	REGION J1.11.1
	    //J1.11.1
	    #"J1.11.1"(ConveyorID := _."J1.11.1",
	               ConveyorSensor:=_."ASiGW-MCC001-bw143-C1: Input"."Sensor J1.11.7",
	               Fault := DB_UDI.EmptyLine.Fault.Stop.Conveyor[_."J1.11.1"],
	               Upstream := DB_UDI.EmptyLine.Upstream.Conveyor[_."J1.11.1"],
	               Downstream := DB_UDI.EmptyLine.DownstreamAcu.Stop.Conveyor[_."J1.11.1"],
	               Interlock := DB_UDI.EmptyLine.Interlock.Stop.Conveyor[_."J1.11.1"],
	               RunForward => _."ASiGW-MCC001-bw143-C1: Output"."Motor J1.11.1",
	               WriteAsiDir => _."ASiGW-MCC001-bw143-C1: Output"."Dir J1.11.1");
	    
	END_REGION
	
	REGION J1.11.2
	    //J1.11.2
	    #"J1.11.2"(ConveyorID:=_."J1.11.2",
	               ConveyorSensor:=_."ASiGW-MCC001-bw143-C1: Input"."Sensor J1.11.7",
	                   Fault:= DB_UDI.EmptyLine.Fault.Stop.Conveyor[_."J1.11.2"],
	                   Upstream:= DB_UDI.EmptyLine.Upstream.Conveyor[_."J1.11.2"],
	                   Downstream:= DB_UDI.EmptyLine.DownstreamAcu.Stop.Conveyor[_."J1.11.2"],
	                   Interlock:= DB_UDI.EmptyLine.Interlock.Stop.Conveyor[_."J1.11.2"],
	                   RunForward => _."ASiGW-MCC001-bw143-C1: Output"."Motor J1.11.2",
	                   WriteAsiDir => _."ASiGW-MCC001-bw143-C1: Output"."Dir J1.11.2");
	
	END_REGION
	
	REGION J1.11.3
	    //J1.11.3
	    #"J1.11.3"(ConveyorID:=_."J1.11.3",
	               ConveyorSensor:=_."ASiGW-MCC001-bw143-C1: Input"."Sensor J1.11.7",
	                   Fault:= DB_UDI.EmptyLine.Fault.Stop.Conveyor[_."J1.11.3"],
	                   Upstream:= DB_UDI.EmptyLine.Upstream.Conveyor[_."J1.11.3"],
	                   Downstream:= DB_UDI.EmptyLine.DownstreamAcu.Stop.Conveyor[_."J1.11.3"],
	                   Interlock:= DB_UDI.EmptyLine.Interlock.Stop.Conveyor[_."J1.11.3"],
	                   RunForward => _."ASiGW-MCC001-bw143-C1: Output"."Motor J1.11.3",
	                   WriteAsiDir => _."ASiGW-MCC001-bw143-C1: Output"."Dir J1.11.3");
	
	END_REGION
	
	REGION J1.11.4
	    //J1.11.4
	    #"J1.11.4"(ConveyorID := _."J1.11.4",
	               ConveyorSensor:=_."ASiGW-MCC001-bw143-C1: Input"."Sensor J1.11.7",
	               Fault := DB_UDI.EmptyLine.Fault.Stop.Conveyor[_."J1.11.4"],
	               Upstream := DB_UDI.EmptyLine.Upstream.Conveyor[_."J1.11.4"],
	               Downstream := DB_UDI.EmptyLine.DownstreamAcu.Stop.Conveyor[_."J1.11.4"],
	               Interlock := DB_UDI.EmptyLine.Interlock.Stop.Conveyor[_."J1.11.4"],
	               RunForward => _."ASiGW-MCC001-bw143-C1: Output"."Motor J1.11.4",
	               WriteAsiDir => _."ASiGW-MCC001-bw143-C1: Output"."Dir J1.11.4");
	    
	END_REGION
	
	REGION J1.11.5
	    //J1.11.5
	    #"J1.11.5"(ConveyorID:=_."J1.11.5",
	               ConveyorSensor:=_."ASiGW-MCC001-bw143-C1: Input"."Sensor J1.11.7",
	                   Fault:= DB_UDI.EmptyLine.Fault.Stop.Conveyor[_."J1.11.5"],
	                   Upstream:= DB_UDI.EmptyLine.Upstream.Conveyor[_."J1.11.5"],
	                   Downstream:= DB_UDI.EmptyLine.DownstreamAcu.Stop.Conveyor[_."J1.11.5"],
	                   Interlock:= DB_UDI.EmptyLine.Interlock.Stop.Conveyor[_."J1.11.5"],
	                   RunForward => _."ASiGW-MCC001-bw143-C1: Output"."Motor J1.11.5",
	                   WriteAsiDir => _."ASiGW-MCC001-bw143-C1: Output"."Dir J1.11.5");
	
	END_REGION
	
	REGION J1.11.6
	    //J1.11.6
	    #"J1.11.6"(ConveyorID := _."J1.11.6",
	               ConveyorSensor:=_."ASiGW-MCC001-bw143-C1: Input"."Sensor J1.11.7",
	               Fault := DB_UDI.EmptyLine.Fault.Stop.Conveyor[_."J1.11.6"],
	               Upstream := DB_UDI.EmptyLine.Upstream.Conveyor[_."J1.11.6"],
	               Downstream := DB_UDI.EmptyLine.DownstreamAcu.Stop.Conveyor[_."J1.11.6"],
	               Interlock := DB_UDI.EmptyLine.Interlock.Stop.Conveyor[_."J1.11.6"],
	               RunForward => _."ASiGW-MCC001-bw143-C1: Output"."Motor J1.11.6",
	               WriteAsiDir => _."ASiGW-MCC001-bw143-C1: Output"."Dir J1.11.6");
	    
	END_REGION
	
	REGION J1.11.7
	    //J1.11.7
	    #"J1.11.7"(ConveyorID := _."J1.11.7",
	               ConveyorSensor:=_."ASiGW-MCC001-bw143-C1: Input"."Sensor J1.11.7",
	               Fault := DB_UDI.EmptyLine.Fault.Stop.Conveyor[_."J1.11.7"],
	               Upstream := DB_UDI.EmptyLine.Upstream.Conveyor[_."J1.11.7"],
	               Downstream := DB_UDI.EmptyLine.DownstreamAcu.Stop.Conveyor[_."J1.11.7"],
	               Interlock := DB_UDI.EmptyLine.Interlock.Stop.Conveyor[_."J1.11.7"],
	               RunForward => _."ASiGW-MCC001-bw143-C1: Output"."Motor J1.11.9",
	               WriteAsiDir => _."ASiGW-MCC001-bw143-C1: Output"."Dir J1.11.9");
	    
	END_REGION
	
	REGION J1.11.8
	    //J1.11.8
	    #"J1.11.8"(ConveyorID := _."J1.11.8",
	               ConveyorSensor:=_."ASiGW-MCC001-bw143-C1: Input"."Sensor J1.11.13",
	               Fault := DB_UDI.EmptyLine.Fault.Stop.Conveyor[_."J1.11.8"],
	               Upstream := DB_UDI.EmptyLine.Upstream.Conveyor[_."J1.11.8"],
	               Downstream := DB_UDI.EmptyLine.DownstreamAcu.Stop.Conveyor[_."J1.11.8"],
	               Interlock := DB_UDI.EmptyLine.Interlock.Stop.Conveyor[_."J1.11.8"],
	               RunForward => _."ASiGW-MCC001-bw143-C1: Output"."Motor J1.11.10",
	               WriteAsiDir => _."ASiGW-MCC001-bw143-C1: Output"."Dir J1.11.10");
	    
	END_REGION
	
	REGION J1.11.9
	    //J1.11.9
	    #"J1.11.9"(ConveyorID:=_."J1.11.9",
	               ConveyorSensor:=_."ASiGW-MCC001-bw143-C1: Input"."Sensor J1.11.13",
	                   Fault:= DB_UDI.EmptyLine.Fault.Stop.Conveyor[_."J1.11.9"],
	                   Upstream:= DB_UDI.EmptyLine.Upstream.Conveyor[_."J1.11.9"],
	                   Downstream:= DB_UDI.EmptyLine.DownstreamAcu.Stop.Conveyor[_."J1.11.9"],
	                   Interlock:= DB_UDI.EmptyLine.Interlock.Stop.Conveyor[_."J1.11.9"],
	                   RunForward => _."ASiGW-MCC001-bw143-C1: Output"."Motor J1.11.11",
	                   WriteAsiDir => _."ASiGW-MCC001-bw143-C1: Output"."Dir J1.11.11");
	        
	END_REGION
	
	REGION J1.11.10
	    //J1.11.10
	    #"J1.11.10"(ConveyorID:=_."J1.11.10",
	                ConveyorSensor:=_."ASiGW-MCC001-bw143-C1: Input"."Sensor J1.11.13",
	                   Fault:= DB_UDI.EmptyLine.Fault.Stop.Conveyor[_."J1.11.10"],
	                   Upstream:= DB_UDI.EmptyLine.Upstream.Conveyor[_."J1.11.10"],
	                   Downstream:= DB_UDI.EmptyLine.DownstreamAcu.Stop.Conveyor[_."J1.11.10"],
	                   Interlock:= DB_UDI.EmptyLine.Interlock.Stop.Conveyor[_."J1.11.10"],
	                   RunForward => _."ASiGW-MCC001-bw143-C1: Output"."Motor J1.11.12",
	                   WriteAsiDir => _."ASiGW-MCC001-bw143-C1: Output"."Dir J1.11.12");
	
	END_REGION
	
	REGION J1.11.11
	    //J1.11.11
	    #"J1.11.11"(ConveyorID:=_."J1.11.11",
	                ConveyorSensor:=_."ASiGW-MCC001-bw143-C1: Input"."Sensor J1.11.13",
	                   Fault:= DB_UDI.EmptyLine.Fault.Stop.Conveyor[_."J1.11.11"],
	                   Upstream:= DB_UDI.EmptyLine.Upstream.Conveyor[_."J1.11.11"],
	                   Downstream:= DB_UDI.EmptyLine.DownstreamAcu.Stop.Conveyor[_."J1.11.11"],
	                   Interlock:= DB_UDI.EmptyLine.Interlock.Stop.Conveyor[_."J1.11.11"],
	                   RunForward => _."ASiGW-MCC001-bw143-C1: Output"."Motor J1.11.13",
	                   WriteAsiDir => _."ASiGW-MCC001-bw143-C1: Output"."Dir J1.11.13");
	
	END_REGION
	
	REGION J1.11.12
	    //J1.11.12
	    #"J1.11.12"(ConveyorID := _."J1.11.12",
	                ConveyorSensor:=_."ASiGW-MCC001-bw143-C1: Input"."Sensor J1.11.13",
	                Fault := DB_UDI.EmptyLine.Fault.Stop.Conveyor[_."J1.11.12"],
	                Upstream := DB_UDI.EmptyLine.Upstream.Conveyor[_."J1.11.12"],
	                Downstream := DB_UDI.EmptyLine.DownstreamAcu.Stop.Conveyor[_."J1.11.12"],
	                Interlock := DB_UDI.EmptyLine.Interlock.Stop.Conveyor[_."J1.11.12"],
	                RunForward => _."ASiGW-MCC001-bw143-C1: Output"."Motor J1.11.12",
	                WriteAsiDir => _."ASiGW-MCC001-bw143-C1: Output"."Dir J1.11.12");
	    
	END_REGION
	
	REGION J1.11.13
	    //J1.11.13
	    #"J1.11.13"(ConveyorID:=_."J1.11.13",
	                ConveyorSensor:=_."ASiGW-MCC001-bw143-C1: Input"."Sensor J1.11.13",
	                   Fault:= DB_UDI.EmptyLine.Fault.Stop.Conveyor[_."J1.11.13"],
	                   Upstream:= DB_UDI.EmptyLine.Upstream.Conveyor[_."J1.11.13"],
	                   Downstream:= DB_UDI.EmptyLine.DownstreamAcu.Stop.Conveyor[_."J1.11.13"],
	                   Interlock:= DB_UDI.EmptyLine.Interlock.Stop.Conveyor[_."J1.11.13"],
	                   RunForward => _."ASiGW-MCC001-bw143-C1: Output"."Motor J1.11.13",
	                   WriteAsiDir => _."ASiGW-MCC001-bw143-C1: Output"."Dir J1.11.13");
	
	END_REGION
	
	REGION K1.1.1
	    //K1.1.1  (Go Left)
	    #"K1.1.1"(ConveyorID:=_."K1.1.1",
	              ConveyorSensor:=_."ASiGW-MCC001-bw143-C2: Input"."Sensor K1.2.1",
	                   Fault:= DB_UDI.EmptyLine.Fault.Stop.Conveyor[_."K1.1.1"],
	                   Upstream:= DB_UDI.EmptyLine.Upstream.Conveyor[_."K1.1.1"],
	                   Downstream:= DB_UDI.EmptyLine.DownstreamAcu.Stop.Conveyor[_."K1.1.1"],
	                   Interlock:= DB_UDI.EmptyLine.Interlock.Stop.Conveyor[_."K1.1.1"],
	                   RunForward => _."ASiGW-MCC001-bw143-C2: Output"."Motor K1.1.1",
	                   WriteAsiDir => _."ASiGW-MCC001-bw143-C2: Output"."Dir K1.1.1");
	         
	END_REGION
	
	REGION K1.2.1
	    //K1.2.1
	    #"K1.2.1"(ConveyorID:=_."K1.2.1",
	              ConveyorSensor:=_."ASiGW-MCC001-bw143-C2: Input"."Sensor K1.2.1",
	                   Fault:= DB_UDI.EmptyLine.Fault.Stop.Conveyor[_."K1.2.1"],
	                   Upstream:= DB_UDI.EmptyLine.Upstream.Conveyor[_."K1.2.1"],
	                   Downstream:= DB_UDI.EmptyLine.DownstreamAcu.Stop.Conveyor[_."K1.2.1"],
	                   Interlock:= DB_UDI.EmptyLine.Interlock.Stop.Conveyor[_."K1.2.1"],
	                   RunForward => _."ASiGW-MCC001-bw143-C2: Output"."Motor - K1.2.1",
	                   WriteAsiDir => _."ASiGW-MCC001-bw143-C2: Output"."2-31A Dir",
	                   WriteAsiSpeed=>_."ASiGW-MCC001-bw143-C2: Output"."2-31A Speed");
	         
	END_REGION
	
	REGION K1.3.1
	    //K1.3.1
	    #"K1.3.1"(ConveyorID := _."K1.3.1",
	              ConveyorSensor:=_."ASiGW-MCC001-bw143-C2: Input"."Sensor K1.3.1",
	              Fault := DB_UDI.EmptyLine.Fault.Stop.Conveyor[_."K1.3.1"],
	              Upstream := DB_UDI.EmptyLine.Upstream.Conveyor[_."K1.3.1"],
	              Downstream := DB_UDI.EmptyLine.DownstreamAcu.Stop.Conveyor[_."K1.3.1"],
	              Interlock := DB_UDI.EmptyLine.Interlock.Stop.Conveyor[_."K1.3.1"],
	              RunForward => _."ASiGW-MCC001-bw143-C2: Output"."Motor K1.3.1",
	              WriteAsiDir => _."ASiGW-MCC001-bw143-C2: Output"."Dir K1.3.1");
	    
	END_REGION
	
	REGION K1.4.1
	    //K1.4.1
	    #"K1.4.1"(ConveyorID:=_."K1.4.1",
	              ConveyorSensor:=_."ASiGW-MCC001-bw143-C2: Input"."Sensor K1.4.1",
	                   Fault:= DB_UDI.EmptyLine.Fault.Stop.Conveyor[_."K1.4.1"],
	                   Upstream:= DB_UDI.EmptyLine.Upstream.Conveyor[_."K1.4.1"],
	                   Downstream:= DB_UDI.EmptyLine.DownstreamAcu.Stop.Conveyor[_."K1.4.1"],
	                   Interlock:= DB_UDI.EmptyLine.Interlock.Stop.Conveyor[_."K1.4.1"],
	                   RunForward => _."ASiGW-MCC001-bw143-C2: Output"."Motor K1.4.1",
	                   WriteAsiDir => _."ASiGW-MCC001-bw143-C2: Output"."Dir K1.4.1");
	         
	END_REGION
	
	REGION K1.4.2
	    //K1.4.2
	    #"K1.4.2"(ConveyorID := _."K1.4.2",
	              ConveyorSensor:=_."ASiGW-MCC001-bw143-C2: Input"."Sensor K1.4.10",
	              Fault := DB_UDI.EmptyLine.Fault.Stop.Conveyor[_."K1.4.2"],
	              Upstream := DB_UDI.EmptyLine.Upstream.Conveyor[_."K1.4.2"],
	              Downstream := DB_UDI.EmptyLine.DownstreamAcu.Stop.Conveyor[_."K1.4.2"],
	              Interlock := DB_UDI.EmptyLine.Interlock.Stop.Conveyor[_."K1.4.2"],
	              RunForward => _."ASiGW-MCC001-bw143-C2: Output"."Motor K1.4.2",
	              WriteAsiDir => _."ASiGW-MCC001-bw143-C2: Output"."Dir K1.4.2");
	    
	END_REGION
	
	REGION K1.4.3
	    //K1.4.3
	    #"K1.4.3"(ConveyorID := _."K1.4.3",
	              ConveyorSensor:=_."ASiGW-MCC001-bw143-C2: Input"."Sensor K1.4.10",
	              Fault := DB_UDI.EmptyLine.Fault.Stop.Conveyor[_."K1.4.3"],
	              Upstream := DB_UDI.EmptyLine.Upstream.Conveyor[_."K1.4.3"],
	              Downstream := DB_UDI.EmptyLine.DownstreamAcu.Stop.Conveyor[_."K1.4.3"],
	              Interlock := DB_UDI.EmptyLine.Interlock.Stop.Conveyor[_."K1.4.3"],
	              RunForward => _."ASiGW-MCC001-bw143-C2: Output"."Motor K1.4.3",
	              WriteAsiDir => _."ASiGW-MCC001-bw143-C2: Output"."Dir K1.4.3");
	    
	END_REGION
	
	REGION K1.4.4
	    //K1.4.4
	    #"K1.4.4"(ConveyorID := _."K1.4.4",
	              ConveyorSensor:=_."ASiGW-MCC001-bw143-C2: Input"."Sensor K1.4.10",
	              Fault := DB_UDI.EmptyLine.Fault.Stop.Conveyor[_."K1.4.4"],
	              Upstream := DB_UDI.EmptyLine.Upstream.Conveyor[_."K1.4.4"],
	              Downstream := DB_UDI.EmptyLine.DownstreamAcu.Stop.Conveyor[_."K1.4.4"],
	              Interlock := DB_UDI.EmptyLine.Interlock.Stop.Conveyor[_."K1.4.4"],
	              RunForward => _."ASiGW-MCC001-bw143-C2: Output"."Motor K1.4.4",
	              WriteAsiDir => _."ASiGW-MCC001-bw143-C2: Output"."Dir K1.4.4");
	    
	END_REGION
	
	REGION K1.4.5
	    //K1.4.5
	    #"K1.4.5"(ConveyorID := _."K1.4.5",
	              ConveyorSensor:=_."ASiGW-MCC001-bw143-C2: Input"."Sensor K1.4.10",
	              Fault := DB_UDI.EmptyLine.Fault.Stop.Conveyor[_."K1.4.5"],
	              Upstream := DB_UDI.EmptyLine.Upstream.Conveyor[_."K1.4.5"],
	              Downstream := DB_UDI.EmptyLine.DownstreamAcu.Stop.Conveyor[_."K1.4.5"],
	              Interlock := DB_UDI.EmptyLine.Interlock.Stop.Conveyor[_."K1.4.5"],
	              RunForward => _."ASiGW-MCC001-bw143-C2: Output"."Motor K1.4.5",
	              WriteAsiDir => _."ASiGW-MCC001-bw143-C2: Output"."Dir K1.4.5");
	    
	END_REGION
	
	REGION K1.4.6
	    //K1.4.6
	    #"K1.4.6"(ConveyorID:=_."K1.4.6",
	              ConveyorSensor:=_."ASiGW-MCC001-bw143-C2: Input"."Sensor K1.4.10",
	                   Fault:= DB_UDI.EmptyLine.Fault.Stop.Conveyor[_."K1.4.6"],
	                   Upstream:= DB_UDI.EmptyLine.Upstream.Conveyor[_."K1.4.6"],
	                   Downstream:= DB_UDI.EmptyLine.DownstreamAcu.Stop.Conveyor[_."K1.4.6"],
	                   Interlock:= DB_UDI.EmptyLine.Interlock.Stop.Conveyor[_."K1.4.6"],
	                   RunForward => _."ASiGW-MCC001-bw143-C2: Output"."Motor K1.4.6",
	                   WriteAsiDir => _."ASiGW-MCC001-bw143-C2: Output"."Dir K1.4.6");
	         
	END_REGION
	
	REGION K1.4.7
	    //K1.4.7
	    #"K1.4.7"(ConveyorID := _."K1.4.7",
	              ConveyorSensor:=_."ASiGW-MCC001-bw143-C2: Input"."Sensor K1.4.10",
	              Fault := DB_UDI.EmptyLine.Fault.Stop.Conveyor[_."K1.4.7"],
	              Upstream := DB_UDI.EmptyLine.Upstream.Conveyor[_."K1.4.7"],
	              Downstream := DB_UDI.EmptyLine.DownstreamAcu.Stop.Conveyor[_."K1.4.7"],
	              Interlock := DB_UDI.EmptyLine.Interlock.Stop.Conveyor[_."K1.4.7"],
	              RunForward => _."ASiGW-MCC001-bw143-C2: Output"."Motor K1.4.7",
	              WriteAsiDir => _."ASiGW-MCC001-bw143-C2: Output"."Dir K1.4.7");
	    
	END_REGION
	
	REGION K1.4.8
	    //K1.4.8
	    #"K1.4.8"(ConveyorID := _."K1.4.8",
	              ConveyorSensor:=_."ASiGW-MCC001-bw143-C2: Input"."Sensor K1.4.10",
	              Fault := DB_UDI.EmptyLine.Fault.Stop.Conveyor[_."K1.4.8"],
	              Upstream := DB_UDI.EmptyLine.Upstream.Conveyor[_."K1.4.8"],
	              Downstream := DB_UDI.EmptyLine.DownstreamAcu.Stop.Conveyor[_."K1.4.8"],
	              Interlock := DB_UDI.EmptyLine.Interlock.Stop.Conveyor[_."K1.4.8"],
	              RunForward => _."ASiGW-MCC001-bw143-C2: Output"."Motor K1.4.8",
	              WriteAsiDir => _."ASiGW-MCC001-bw143-C2: Output"."Dir K1.4.8");
	    
	END_REGION
	
	REGION K1.4.9
	    //K1.4.9
	    #"K1.4.9"(ConveyorID:=_."K1.4.9",
	              ConveyorSensor:=_."ASiGW-MCC001-bw143-C2: Input"."Sensor K1.4.10",
	                   Fault:= DB_UDI.EmptyLine.Fault.Stop.Conveyor[_."K1.4.9"],
	                   Upstream:= DB_UDI.EmptyLine.Upstream.Conveyor[_."K1.4.9"],
	                   Downstream:= DB_UDI.EmptyLine.DownstreamAcu.Stop.Conveyor[_."K1.4.9"],
	                   Interlock:= DB_UDI.EmptyLine.Interlock.Stop.Conveyor[_."K1.4.9"],
	                   RunForward => _."ASiGW-MCC001-bw143-C2: Output"."Motor K1.4.9",
	                   WriteAsiDir => _."ASiGW-MCC001-bw143-C2: Output"."Dir K1.4.9");
	         
	END_REGION
	
	REGION K1.4.10
	    //K1.4.10
	    #"K1.4.10"(ConveyorID:=_."K1.4.10",
	               ConveyorSensor:=_."ASiGW-MCC001-bw143-C2: Input"."Sensor K1.4.10",
	                   Fault:= DB_UDI.EmptyLine.Fault.Stop.Conveyor[_."K1.4.10"],
	                   Upstream:= DB_UDI.EmptyLine.Upstream.Conveyor[_."K1.4.10"],
	                   Downstream:= DB_UDI.EmptyLine.DownstreamAcu.Stop.Conveyor[_."K1.4.10"],
	                   Interlock:= DB_UDI.EmptyLine.Interlock.Stop.Conveyor[_."K1.4.10"],
	                   RunForward => _."ASiGW-MCC001-bw143-C2: Output"."Motor K1.4.10",
	                   WriteAsiDir => _."ASiGW-MCC001-bw143-C2: Output"."Dir K1.4.10");
	        
	END_REGION
	
	REGION K1.5.1
	    //K1.5.1
	    #"K1.5.1"(ConveyorID:=_."K1.5.1",
	              ConveyorSensor:=_."ASiGW-MCC001-bw143-C2: Input"."Sensor K1.5.8",
	                   Fault:= DB_UDI.EmptyLine.Fault.Stop.Conveyor[_."K1.5.1"],
	                   Upstream:= DB_UDI.EmptyLine.Upstream.Conveyor[_."K1.5.1"],
	                   Downstream:= DB_UDI.EmptyLine.DownstreamAcu.Stop.Conveyor[_."K1.5.1"],
	                   Interlock:= DB_UDI.EmptyLine.Interlock.Stop.Conveyor[_."K1.5.1"],
	                   RunForward => _."ASiGW-MCC001-bw143-C2: Output"."Motor K1.5.1",
	                   WriteAsiDir => _."ASiGW-MCC001-bw143-C2: Output"."Dir K1.5.1");
	
	END_REGION
	
	REGION K1.5.2
	    //K1.5.2
	    #"K1.5.2"(ConveyorID:=_."K1.5.2",
	              ConveyorSensor:=_."ASiGW-MCC001-bw143-C2: Input"."Sensor K1.5.8",
	                   Fault:= DB_UDI.EmptyLine.Fault.Stop.Conveyor[_."K1.5.2"],
	                   Upstream:= DB_UDI.EmptyLine.Upstream.Conveyor[_."K1.5.2"],
	                   Downstream:= DB_UDI.EmptyLine.DownstreamAcu.Stop.Conveyor[_."K1.5.2"],
	                   Interlock:= DB_UDI.EmptyLine.Interlock.Stop.Conveyor[_."K1.5.2"],
	                   RunForward => _."ASiGW-MCC001-bw143-C2: Output"."Motor K1.5.2",
	                   WriteAsiDir => _."ASiGW-MCC001-bw143-C2: Output"."Dir K1.5.2");
	         
	
	END_REGION
	
	REGION K1.5.3
	    //K1.5.3
	    #"K1.5.3"(ConveyorID:=_."K1.5.3",
	              ConveyorSensor:=_."ASiGW-MCC001-bw143-C2: Input"."Sensor K1.5.8",
	                   Fault:= DB_UDI.EmptyLine.Fault.Stop.Conveyor[_."K1.5.3"],
	                   Upstream:= DB_UDI.EmptyLine.Upstream.Conveyor[_."K1.5.3"],
	                   Downstream:= DB_UDI.EmptyLine.DownstreamAcu.Stop.Conveyor[_."K1.5.3"],
	                   Interlock:= DB_UDI.EmptyLine.Interlock.Stop.Conveyor[_."K1.5.3"],
	                   RunForward => _."ASiGW-MCC001-bw143-C2: Output"."Motor K1.5.3",
	                   WriteAsiDir => _."ASiGW-MCC001-bw143-C2: Output"."Dir K1.5.3");
	         
	
	END_REGION
	
	REGION K1.5.4
	    //K1.5.4
	    #"K1.5.4"(ConveyorID:=_."K1.5.4",
	              ConveyorSensor:=_."ASiGW-MCC001-bw143-C2: Input"."Sensor K1.5.8",
	                   Fault:= DB_UDI.EmptyLine.Fault.Stop.Conveyor[_."K1.5.4"],
	                   Upstream:= DB_UDI.EmptyLine.Upstream.Conveyor[_."K1.5.4"],
	                   Downstream:= DB_UDI.EmptyLine.DownstreamAcu.Stop.Conveyor[_."K1.5.4"],
	                   Interlock:= DB_UDI.EmptyLine.Interlock.Stop.Conveyor[_."K1.5.4"],
	                   RunForward => _."ASiGW-MCC001-bw143-C2: Output"."Motor K1.5.4",
	                   WriteAsiDir => _."ASiGW-MCC001-bw143-C2: Output"."Dir K1.5.4");
	         
	END_REGION
	
	REGION K1.5.5
	    //K1.5.5
	    #"K1.5.5"(ConveyorID := _."K1.5.5",
	              ConveyorSensor:=_."ASiGW-MCC001-bw143-C2: Input"."Sensor K1.5.8",
	              Fault := DB_UDI.EmptyLine.Fault.Stop.Conveyor[_."K1.5.5"],
	              Upstream := DB_UDI.EmptyLine.Upstream.Conveyor[_."K1.5.5"],
	              Downstream := DB_UDI.EmptyLine.DownstreamAcu.Stop.Conveyor[_."K1.5.5"],
	              Interlock := DB_UDI.EmptyLine.Interlock.Stop.Conveyor[_."K1.5.5"],
	              RunForward => _."ASiGW-MCC001-bw143-C2: Output"."Motor K1.5.5",
	              WriteAsiDir => _."ASiGW-MCC001-bw143-C2: Output"."Dir K1.5.5");
	    
	    
	END_REGION
	
	REGION K1.5.6
	    //K1.5.6
	    #"K1.5.6"(ConveyorID:=_."K1.5.6",
	              ConveyorSensor:=_."ASiGW-MCC001-bw143-C2: Input"."Sensor K1.5.8",
	                   Fault:= DB_UDI.EmptyLine.Fault.Stop.Conveyor[_."K1.5.6"],
	                   Upstream:= DB_UDI.EmptyLine.Upstream.Conveyor[_."K1.5.6"],
	                   Downstream:= DB_UDI.EmptyLine.DownstreamAcu.Stop.Conveyor[_."K1.5.6"],
	                   Interlock:= DB_UDI.EmptyLine.Interlock.Stop.Conveyor[_."K1.5.6"],
	                   RunForward => _."ASiGW-MCC001-bw143-C2: Output"."Motor K1.5.6",
	                   WriteAsiDir => _."ASiGW-MCC001-bw143-C2: Output"."Dir K1.5.6");
	        
	
	END_REGION
	
	REGION K1.5.7
	    //K1.5.7
	    #"K1.5.7"(ConveyorID:=_."K1.5.7",
	              ConveyorSensor:=_."ASiGW-MCC001-bw143-C2: Input"."Sensor K1.5.8",
	                   Fault:= DB_UDI.EmptyLine.Fault.Stop.Conveyor[_."K1.5.7"],
	                   Upstream:= DB_UDI.EmptyLine.Upstream.Conveyor[_."K1.5.7"],
	                   Downstream:= DB_UDI.EmptyLine.DownstreamAcu.Stop.Conveyor[_."K1.5.7"],
	                   Interlock:= DB_UDI.EmptyLine.Interlock.Stop.Conveyor[_."K1.5.7"],
	                   RunForward => _."ASiGW-MCC001-bw143-C2: Output"."Motor K1.5.7",
	                   WriteAsiDir => _."ASiGW-MCC001-bw143-C2: Output"."Dir K1.5.7");
	         
	END_REGION
	
	REGION K1.5.8
	    //K1.5.8
	    #"K1.5.8"(ConveyorID:=_."K1.5.8",
	              ConveyorSensor:=_."ASiGW-MCC001-bw143-C2: Input"."Sensor K1.5.8",
	                   Fault:= DB_UDI.EmptyLine.Fault.Stop.Conveyor[_."K1.5.8"],
	                   Upstream:= DB_UDI.EmptyLine.Upstream.Conveyor[_."K1.5.8"],
	                   Downstream:= DB_UDI.EmptyLine.DownstreamAcu.Stop.Conveyor[_."K1.5.8"],
	                   Interlock:= DB_UDI.EmptyLine.Interlock.Stop.Conveyor[_."K1.5.8"],
	                   RunForward => _."ASiGW-MCC001-bw143-C2: Output"."Motor K1.5.8",
	                   WriteAsiDir => _."ASiGW-MCC001-bw143-C2: Output"."Dir K1.5.8");
	         
	END_REGION
	
	REGION K1.6.1
	    //K1.6.1
	    #"K1.6.1"(ConveyorID:=_."K1.6.1",
	              ConveyorSensor:=_."ASiGW-MCC001-bw143-C2: Input"."Sensor K1.6.1",
	                   Fault:= DB_UDI.EmptyLine.Fault.Stop.Conveyor[_."K1.6.1"],
	                   Upstream:= DB_UDI.EmptyLine.Upstream.Conveyor[_."K1.6.1"],
	                   Downstream:= DB_UDI.EmptyLine.DownstreamAcu.Stop.Conveyor[_."K1.6.1"],
	                   Interlock:= DB_UDI.EmptyLine.Interlock.Stop.Conveyor[_."K1.6.1"],
	                   RunForward => _."ASiGW-MCC001-bw143-C2: Output"."Motor - K1.6.1",
	                   WriteAsiDir => _."ASiGW-MCC001-bw143-C2: Output"."2-11B Dir",
	                   WriteAsiSpeed=> _."ASiGW-MCC001-bw143-C2: Output"."2-11B Speed");
	         
	END_REGION
	
	REGION K1.6.2
	    //K1.6.2
	    #"K1.6.2"(ConveyorID := _."K1.6.2",
	              ConveyorSensor:=_."ASiGW-MCC001-bw143-C2: Input"."Sensor K1.6.2",
	              Fault := DB_UDI.EmptyLine.Fault.Stop.Conveyor[_."K1.6.2"],
	              Upstream := DB_UDI.EmptyLine.Upstream.Conveyor[_."K1.6.2"],
	              Downstream := DB_UDI.EmptyLine.DownstreamAcu.Stop.Conveyor[_."K1.6.2"],
	              Interlock := DB_UDI.EmptyLine.Interlock.Stop.Conveyor[_."K1.6.2"],
	              RunForward => _."ASiGW-MCC001-bw143-C2: Output"."Motor - K1.6.2",
	              WriteAsiDir => _."ASiGW-MCC001-bw143-C2: Output"."2-11B Dir",
	              WriteAsiSpeed => _."ASiGW-MCC001-bw143-C2: Output"."2-11B Speed");
	    
	END_REGION
	
	REGION K1.7.1
	    //K1.7.1
	    #"K1.7.1"(ConveyorID := _."K1.7.1",
	              ConveyorSensor:=_."ASiGW-MCC001-bw143-C2: Input"."Sensor K1.7.2",
	              Fault := DB_UDI.EmptyLine.Fault.Stop.Conveyor[_."K1.7.1"],
	              Upstream := DB_UDI.EmptyLine.Upstream.Conveyor[_."K1.7.1"],
	              Downstream := DB_UDI.EmptyLine.DownstreamAcu.Stop.Conveyor[_."K1.7.1"],
	              Interlock := DB_UDI.EmptyLine.Interlock.Stop.Conveyor[_."K1.7.1"],
	              RunForward => _."ASiGW-MCC001-bw143-C2: Output"."Motor K1.7.1",
	              WriteAsiDir => _."ASiGW-MCC001-bw143-C2: Output"."Dir K1.7.1");
	    
	END_REGION
	
	REGION K1.7.2
	    //K1.7.2
	    #"K1.7.2"(ConveyorID := _."K1.7.2",
	              ConveyorSensor:=_."ASiGW-MCC001-bw143-C2: Input"."Sensor K1.7.2",
	              Fault := DB_UDI.EmptyLine.Fault.Stop.Conveyor[_."K1.7.2"],
	              Upstream := DB_UDI.EmptyLine.Upstream.Conveyor[_."K1.7.2"],
	              Downstream := DB_UDI.EmptyLine.DownstreamAcu.Stop.Conveyor[_."K1.7.2"],
	              Interlock := DB_UDI.EmptyLine.Interlock.Stop.Conveyor[_."K1.7.2"],
	              RunForward => _."ASiGW-MCC001-bw143-C2: Output"."Motor K1.7.2",
	              WriteAsiDir => _."ASiGW-MCC001-bw143-C2: Output"."Dir K1.7.2");
	    
	END_REGION
	
	REGION K1.8.1
	    //K1.8.1
	    #"K1.8.1"(ConveyorID:=_."K1.8.1",
	              ConveyorSensor:=_."ASiGW-MCC001-bw143-C2: Input"."Sensor K1.8.3",
	                   Fault:= DB_UDI.EmptyLine.Fault.Stop.Conveyor[_."K1.8.1"],
	                   Upstream:= DB_UDI.EmptyLine.Upstream.Conveyor[_."K1.8.1"],
	                   Downstream:= DB_UDI.EmptyLine.DownstreamAcu.Stop.Conveyor[_."K1.8.1"],
	                   Interlock:= DB_UDI.EmptyLine.Interlock.Stop.Conveyor[_."K1.8.1"],
	                   RunForward => _."ASiGW-MCC001-bw143-C2: Output"."Motor K1.8.1",
	                   WriteAsiDir => _."ASiGW-MCC001-bw143-C2: Output"."Dir K1.8.1");
	
	END_REGION
	
	REGION K1.8.2
	    //K1.8.2
	    #"K1.8.2"(ConveyorID := _."K1.8.2",
	              ConveyorSensor:=_."ASiGW-MCC001-bw143-C2: Input"."Sensor K1.8.3",
	              Fault := DB_UDI.EmptyLine.Fault.Stop.Conveyor[_."K1.8.2"],
	              Upstream := DB_UDI.EmptyLine.Upstream.Conveyor[_."K1.8.2"],
	              Downstream := DB_UDI.EmptyLine.DownstreamAcu.Stop.Conveyor[_."K1.8.2"],
	              Interlock := DB_UDI.EmptyLine.Interlock.Stop.Conveyor[_."K1.8.2"],
	              RunForward => _."ASiGW-MCC001-bw143-C2: Output"."Motor K1.8.2",
	              WriteAsiDir => _."ASiGW-MCC001-bw143-C2: Output"."Dir K1.8.2");
	    
	END_REGION
	
	REGION K1.8.3
	    //K1.8.3
	    #"K1.8.3"(ConveyorID := _."K1.8.3",
	              ConveyorSensor:=_."ASiGW-MCC001-bw143-C2: Input"."Sensor K1.8.3",
	              Fault := DB_UDI.EmptyLine.Fault.Stop.Conveyor[_."K1.8.3"],
	              Upstream := DB_UDI.EmptyLine.Upstream.Conveyor[_."K1.8.3"],
	              Downstream := DB_UDI.EmptyLine.DownstreamAcu.Stop.Conveyor[_."K1.8.3"],
	              Interlock := DB_UDI.EmptyLine.Interlock.Stop.Conveyor[_."K1.8.3"],
	              RunForward => _."ASiGW-MCC001-bw143-C2: Output"."Motor K1.8.3",
	              WriteAsiDir => _."ASiGW-MCC001-bw143-C2: Output"."Dir K1.8.3");
	    
	END_REGION
	
	REGION K1.9.1
	    //K1.9.1
	    #"K1.9.1"(ConveyorID := _."K1.9.1",
	              ConveyorSensor:=_."ASiGW-MCC001-bw143-C2: Input"."Sensor K1.10.1",
	              Fault := DB_UDI.EmptyLine.Fault.Stop.Conveyor[_."K1.9.1"],
	              Upstream := DB_UDI.EmptyLine.Upstream.Conveyor[_."K1.9.1"],
	              Downstream := DB_UDI.EmptyLine.DownstreamAcu.Stop.Conveyor[_."K1.9.1"],
	              Interlock := DB_UDI.EmptyLine.Interlock.Stop.Conveyor[_."K1.9.1"],
	              RunForward => _."ASiGW-MCC001-bw143-C2: Output"."Motor K1.9.1",
	              WriteAsiDir => _."ASiGW-MCC001-bw143-C2: Output"."Dir K1.9.1");
	    
	END_REGION
	
	REGION K1.9.2
	    //K1.9.2
	    #"K1.9.2"(ConveyorID:=_."K1.9.2",
	              ConveyorSensor:=_."ASiGW-MCC001-bw143-C2: Input"."Sensor K1.10.1",
	                   Fault:= DB_UDI.EmptyLine.Fault.Stop.Conveyor[_."K1.9.2"],
	                   Upstream:= DB_UDI.EmptyLine.Upstream.Conveyor[_."K1.9.2"],
	                   Downstream:= DB_UDI.EmptyLine.DownstreamAcu.Stop.Conveyor[_."K1.9.2"],
	                   Interlock:= DB_UDI.EmptyLine.Interlock.Stop.Conveyor[_."K1.9.2"],
	                   RunForward => _."ASiGW-MCC001-bw143-C2: Output"."Motor K1.9.2",
	                   WriteAsiDir => _."ASiGW-MCC001-bw143-C2: Output"."Dir K1.9.3");
	         
	END_REGION
	
	REGION K1.9.3
	    //K1.9.3
	    #"K1.9.3"(ConveyorID := _."K1.9.3",
	              ConveyorSensor:=_."ASiGW-MCC001-bw143-C2: Input"."Sensor K1.10.1",
	              Fault := DB_UDI.EmptyLine.Fault.Stop.Conveyor[_."K1.9.3"],
	              Upstream := DB_UDI.EmptyLine.Upstream.Conveyor[_."K1.9.3"],
	              Downstream := DB_UDI.EmptyLine.DownstreamAcu.Stop.Conveyor[_."K1.9.3"],
	              Interlock := DB_UDI.EmptyLine.Interlock.Stop.Conveyor[_."K1.9.3"],
	              RunForward => _."ASiGW-MCC001-bw143-C2: Output"."Motor K1.9.3",
	              WriteAsiDir => _."ASiGW-MCC001-bw143-C2: Output"."Dir K1.9.3");
	    
	END_REGION
	
	REGION K1.9.4
	    //K1.9.4
	    #"K1.9.4"(ConveyorID := _."K1.9.4",
	              ConveyorSensor:=_."ASiGW-MCC001-bw143-C2: Input"."Sensor K1.10.1",
	              Fault := DB_UDI.EmptyLine.Fault.Stop.Conveyor[_."K1.9.4"],
	              Upstream := DB_UDI.EmptyLine.Upstream.Conveyor[_."K1.9.4"],
	              Downstream := DB_UDI.EmptyLine.DownstreamAcu.Stop.Conveyor[_."K1.9.4"],
	              Interlock := DB_UDI.EmptyLine.Interlock.Stop.Conveyor[_."K1.9.4"],
	              RunForward => _."ASiGW-MCC001-bw143-C2: Output"."Motor K1.9.4",
	              WriteAsiDir => _."ASiGW-MCC001-bw143-C2: Output"."Dir K1.9.4");
	    
	END_REGION
	
	REGION K1.9.5
	    //K1.9.5
	    #"K1.9.5"(ConveyorID := _."K1.9.5",
	              ConveyorSensor:=_."ASiGW-MCC001-bw143-C2: Input"."Sensor K1.10.1",
	              Fault := DB_UDI.EmptyLine.Fault.Stop.Conveyor[_."K1.9.5"],
	              Upstream := DB_UDI.EmptyLine.Upstream.Conveyor[_."K1.9.5"],
	              Downstream := DB_UDI.EmptyLine.DownstreamAcu.Stop.Conveyor[_."K1.9.5"],
	              Interlock := DB_UDI.EmptyLine.Interlock.Stop.Conveyor[_."K1.9.5"],
	              RunForward => _."ASiGW-MCC001-bw143-C2: Output"."Motor K1.9.5",
	              WriteAsiDir => _."ASiGW-MCC001-bw143-C2: Output"."Dir K1.9.5");
	    
	END_REGION
	
	REGION K1.9.6
	    //K1.9.6
	    #"K1.9.6"(ConveyorID := _."K1.9.6",
	              ConveyorSensor:=_."ASiGW-MCC001-bw143-C2: Input"."Sensor K1.10.1",
	              Fault := DB_UDI.EmptyLine.Fault.Stop.Conveyor[_."K1.9.6"],
	              Upstream := DB_UDI.EmptyLine.Upstream.Conveyor[_."K1.9.6"],
	              Downstream := DB_UDI.EmptyLine.DownstreamAcu.Stop.Conveyor[_."K1.9.6"],
	              Interlock := DB_UDI.EmptyLine.Interlock.Stop.Conveyor[_."K1.9.6"],
	              RunForward => _."ASiGW-MCC001-bw143-C2: Output"."Motor K1.9.6",
	              WriteAsiDir => _."ASiGW-MCC001-bw143-C2: Output"."Dir K1.9.6");
	    
	END_REGION
	
	REGION K1.9.7
	    //K1.9.7
	    #"K1.9.7"(ConveyorID:=_."K1.9.7",
	              ConveyorSensor:=_."ASiGW-MCC001-bw143-C2: Input"."Sensor K1.10.1",
	              Fault:= DB_UDI.EmptyLine.Fault.Stop.Conveyor[_."K1.9.7"],
	              Upstream:= DB_UDI.EmptyLine.Upstream.Conveyor[_."K1.9.7"],
	              Downstream:= DB_UDI.EmptyLine.DownstreamAcu.Stop.Conveyor[_."K1.9.7"],
	              Interlock:= DB_UDI.EmptyLine.Interlock.Stop.Conveyor[_."K1.9.7"],
	              RunForward => _."ASiGW-MCC001-bw143-C2: Output"."Motor K1.9.7",
	              WriteAsiDir => _."ASiGW-MCC001-bw143-C2: Output"."Dir K1.9.7");
	END_REGION
	
	REGION K1.10.1
	    //K1.10.1
	    #"K1.10.1"(ConveyorID := _."K1.10.1",
	               ConveyorSensor:=_."ASiGW-MCC001-bw143-C2: Input"."Sensor K1.10.1",
	               Fault := DB_UDI.EmptyLine.Fault.Stop.Conveyor[_."K1.10.1"],
	               Upstream := DB_UDI.EmptyLine.Upstream.Conveyor[_."K1.10.1"],
	               Downstream := DB_UDI.EmptyLine.DownstreamAcu.Stop.Conveyor[_."K1.10.1"],
	               Interlock := DB_UDI.EmptyLine.Interlock.Stop.Conveyor[_."K1.10.1"],
	               RunForward => _."ASiGW-MCC001-bw143-C2: Output"."Motor K1.10.1",
	               WriteAsiDir => _."ASiGW-MCC001-bw143-C2: Output"."Dir K1.10.1");
	    
	END_REGION
	
	
	
	
	
	
	
	
	
	
END_FUNCTION_BLOCK
END_NAMESPACE

NAMESPACE EmptyLine
ORGANIZATION_BLOCK Main_EmptyLine
TITLE = "Main Program Sweep (Cycle)"
{ S7_Optimized_Access := 'TRUE' ; Published := 'FALSE' }
VERSION : 0.1

BEGIN
	// ==========================================================================================================================================
	// Company        : LogTech, s.r.o.
	// Created by     : Anton Vinoth Soundraraj
	// Block          : Main_LineB1
	// Project        : Lékarna DC Chrudim
	// Project number : 23-157
	// ==========================================================================================================================================
	
	IDB_EmptyLine();
	
	IDB_Merging();
	
END_ORGANIZATION_BLOCK
END_NAMESPACE

NAMESPACE Global
FUNCTION_BLOCK FB_GlobalStatus
{ S7_Optimized_Access := 'TRUE' ; Published := 'FALSE' }
VERSION : 0.1
   VAR 
      Line : Struct
         ProductionLine { S7_SetPoint := 'False'} : ConveyorStatus;
         EmptyLine : ConveyorStatus;
         PackedLine : ConveyorStatus;
      END_STRUCT;
      cmp : Struct
         ProductionTotes_Value0 : Array[_.gminProductionLine.._.gmaxProductionLine] of Bool;
         ProductionTotes_Value1 : Array[_.gminProductionLine.._.gmaxProductionLine] of Bool;
         EmptyLine_Value0 : Array[_.gminEmptyLine.._.gmaxEmptyLine] of Bool;
         EmptyLine_Value1 : Array[_.gminEmptyLine.._.gmaxEmptyLine] of Bool;
         PackedLine_Value0 : Array[_.gminPackedLine.._.gmaxPackedLine] of Bool;
         PackedLine_Value1 : Array[_.gminPackedLine.._.gmaxPackedLine] of Bool;
      END_STRUCT;
      ForVisu : Struct
         Line : Struct
            ProductionLine : Word;
            EmptyLine : Word;
            PackedLine : Word;
         END_STRUCT;
      END_STRUCT;
   END_VAR


BEGIN
	// ==========================================================================================================================================
	// Company        : LogTech, s.r.o.
	// Created by     : Anton Vinoth Soundraraj
	// Block          : FB_GlobalStatus
	// Project        : Lékarna DC Chrudim
	// Project number : 23-157
	// ==========================================================================================================================================
	
	REGION Line ProductionTotes
	    
	    REGION Line ProductionLine global status
	        
	        // Blockage
	        // initial status: global BLOCKAGE is deactivated
	        // If any of the conveyor gets BLOCKAGE status; global blockage -> activated 
	        #Line.ProductionLine.Blockage :=
	        NOT (#cmp.ProductionTotes_Value0 = DB_Global.Status.Line.ProductionLine.Blockage);
	        
	        // on
	        // initial status: global ON is activated
	        // If any of the conveyor gets NOT ON status; global ON -> deactivated  
	        #Line.ProductionLine.ON :=
	        (#cmp.ProductionTotes_Value1 = DB_Global.Status.Line.ProductionLine.On);
	        
	        // ready to run
	        // initial status: global READY is activated
	        // If any of the conveyor gets NOT READY status; global ready -> deactivated 
	        #Line.ProductionLine.ReadytoRun :=
	        (#cmp.ProductionTotes_Value1 = DB_Global.Status.Line.ProductionLine.ReadyToRun);
	        
	        // occupied
	        // initial status: global OCCUPIED is activated
	        // If all the conveyor are OCCUPIED; global OCCUPIED -> activated  
	        #Line.ProductionLine.ON :=
	        (#cmp.ProductionTotes_Value1 = DB_Global.Status.Line.ProductionLine.Occupied);
	        
	        // fault
	        // initial status: global FAULT is deactivated
	        // If any of the conveyor gets FAULT status; global fault -> activated
	        #Line.ProductionLine.Fault :=
	        NOT (#cmp.ProductionTotes_Value0 = DB_Global.Status.Line.ProductionLine.Fault);
	        
	        // estop
	        // initial status: global ESTOP is deactivated
	        // If any of the conveyor gets ESTOP status; global estop -> activated
	        #Line.ProductionLine.Estop :=
	        NOT (#cmp.ProductionTotes_Value0 = DB_Global.Status.Line.ProductionLine.Estop);
	        
	        // Manual
	        // initial status: global MANUAL is deactivated
	        // If any of the conveyor gets MANUAL status; global MANUAL -> activated
	        #Line.ProductionLine.Manual :=
	        NOT (#cmp.ProductionTotes_Value0 = DB_Global.Status.Line.ProductionLine.Manual);
	        
	        // stop
	        // initial status: global STOP is deactivated
	        // If any of the conveyor gets STOP status; global stop -> activated
	        #Line.ProductionLine.Stop :=
	        NOT (#cmp.ProductionTotes_Value0 = DB_Global.Status.Line.ProductionLine.Stop);
	        
	    END_REGION
	    
	    REGION Line ProductionLine color for HMI
	        
	        // each and every status of the conveyor will be mentioned by different colors in HMI panel
	        
	        #ForVisu.Line.ProductionLine.%X8 := #Line.ProductionLine.Blockage;
	        #ForVisu.Line.ProductionLine.%X0 := #Line.ProductionLine.ON;
	        #ForVisu.Line.ProductionLine.%X1 := #Line.ProductionLine.ReadytoRun;
	        #ForVisu.Line.ProductionLine.%X2 := #Line.ProductionLine.Occupied;
	        #ForVisu.Line.ProductionLine.%X3 := #Line.ProductionLine.Running;
	        #ForVisu.Line.ProductionLine.%X4 := #Line.ProductionLine.Fault;
	        #ForVisu.Line.ProductionLine.%X5 := #Line.ProductionLine.Estop;
	        #ForVisu.Line.ProductionLine.%X6 := #Line.ProductionLine.Manual;
	        #ForVisu.Line.ProductionLine.%X7 := #Line.ProductionLine.Stop;
	        
	        // convert word to Interger value: 
	        // color will be depends on the status priority (integer value) 
	        // reference: Conveyor image in HMI screen -> property -> Apperance   
	        
	        DB_VisuColor.Line.ProductionLine.GlobalStatus :=
	        WORD_TO_INT(#ForVisu.Line.ProductionLine);
	        
	    END_REGION
	    
	END_REGION
	
	REGION Line EmptyLine
	    
	    REGION Line EmptyLine global status
	        
	        // Blockage
	        // initial status: global BLOCKAGE is deactivated
	        // If any of the conveyor gets BLOCKAGE status; global blockage -> activated 
	        #Line.EmptyLine.Blockage :=
	        NOT (#cmp.EmptyLine_Value0 =DB_Global.Status.Line.EmptyLine.Blockage);
	        
	        // on
	        // initial status: global ON is activated
	        // If any of the conveyor gets NOT ON status; global ON -> deactivated  
	        #Line.EmptyLine.ON :=
	        (#cmp.EmptyLine_Value1 = DB_Global.Status.Line.EmptyLine.On);
	        
	        // ready to run
	        // initial status: global READY is activated
	        // If any of the conveyor gets NOT READY status; global ready -> deactivated 
	        #Line.EmptyLine.ReadytoRun :=
	        (#cmp.EmptyLine_Value1 = DB_Global.Status.Line.EmptyLine.ReadyToRun);
	        
	        // occupied
	        // initial status: global OCCUPIED is activated
	        // If all the conveyor are OCCUPIED; global OCCUPIED -> activated  
	        #Line.EmptyLine.ON :=
	        (#cmp.EmptyLine_Value1 =DB_Global.Status.Line.EmptyLine.Occupied);
	        
	        // fault
	        // initial status: global FAULT is deactivated
	        // If any of the conveyor gets FAULT status; global fault -> activated
	        #Line.EmptyLine.Fault :=
	        NOT (#cmp.EmptyLine_Value0 = DB_Global.Status.Line.EmptyLine.Fault);
	        
	        // estop
	        // initial status: global ESTOP is deactivated
	        // If any of the conveyor gets ESTOP status; global estop -> activated
	        #Line.EmptyLine.Estop :=
	        NOT (#cmp.EmptyLine_Value0 = DB_Global.Status.Line.EmptyLine.Estop);
	        
	        // Manual
	        // initial status: global MANUAL is deactivated
	        // If any of the conveyor gets MANUAL status; global MANUAL -> activated
	        #Line.EmptyLine.Manual :=
	        NOT (#cmp.EmptyLine_Value0 = DB_Global.Status.Line.EmptyLine.Manual);
	        
	        // stop
	        // initial status: global STOP is deactivated
	        // If any of the conveyor gets STOP status; global stop -> activated
	        #Line.EmptyLine.Stop :=
	        NOT (#cmp.EmptyLine_Value0 = DB_Global.Status.Line.EmptyLine.Stop);
	        
	    END_REGION
	    
	    REGION Line EmptyLine color for HMI
	        
	        // each and every status of the conveyor will be mentioned by different colors in HMI panel
	        
	        #ForVisu.Line.EmptyLine.%X8 := #Line.EmptyLine.Blockage;
	        // for future
	        (* OR
	        "IDB_KeyenceBP-I".TriggerSensorBlocked OR
	        "IDB_HeightSensor".BlockageActive *)
	        #ForVisu.Line.EmptyLine.%X0 := #Line.EmptyLine.ON;
	        #ForVisu.Line.EmptyLine.%X1 := #Line.EmptyLine.ReadytoRun;
	        #ForVisu.Line.EmptyLine.%X2 := #Line.EmptyLine.Occupied;
	        #ForVisu.Line.EmptyLine.%X3 := #Line.EmptyLine.Running;
	        #ForVisu.Line.EmptyLine.%X4 := #Line.EmptyLine.Fault;
	        #ForVisu.Line.EmptyLine.%X5 := #Line.EmptyLine.Estop;
	        #ForVisu.Line.EmptyLine.%X6 := #Line.EmptyLine.Manual;
	        #ForVisu.Line.EmptyLine.%X7 := #Line.EmptyLine.Stop;
	        
	        // convert word to Interger value: 
	        // color will be depends on the status priority (integer value) 
	        // reference: Conveyor image in HMI screen -> property -> Apperance   
	        
	        DB_VisuColor.Line.EmptyLine.GlobalStatus :=
	        WORD_TO_INT(#ForVisu.Line.EmptyLine);
	        
	    END_REGION
	    
	END_REGION
	
	REGION Line PackedLine
	    
	    REGION Line PackedLine global status
	        
	        // Blockage
	        // initial status: global BLOCKAGE is deactivated
	        // If any of the conveyor gets BLOCKAGE status; global blockage -> activated 
	        #Line.PackedLine.Blockage :=
	        NOT (#cmp.PackedLine_Value0 = DB_Global.Status.Line.PackedLine.Blockage);
	        
	        // on
	        // initial status: global ON is activated
	        // If any of the conveyor gets NOT ON status; global ON -> deactivated  
	        #Line.PackedLine.ON :=
	        (#cmp.PackedLine_Value1 = DB_Global.Status.Line.PackedLine.On);
	        
	        // ready to run
	        // initial status: global READY is activated
	        // If any of the conveyor gets NOT READY status; global ready -> deactivated 
	        #Line.PackedLine.ReadytoRun :=
	        (#cmp.PackedLine_Value1 = DB_Global.Status.Line.PackedLine.ReadyToRun);
	        
	        // occupied
	        // initial status: global OCCUPIED is activated
	        // If all the conveyor are OCCUPIED; global OCCUPIED -> activated  
	        #Line.PackedLine.ON :=
	        (#cmp.PackedLine_Value1 = DB_Global.Status.Line.PackedLine.Occupied);
	        
	        // fault
	        // initial status: global FAULT is deactivated
	        // If any of the conveyor gets FAULT status; global fault -> activated
	        #Line.PackedLine.Fault :=
	        NOT (#cmp.PackedLine_Value0 = DB_Global.Status.Line.PackedLine.Fault);
	        
	        // estop
	        // initial status: global ESTOP is deactivated
	        // If any of the conveyor gets ESTOP status; global estop -> activated
	        #Line.PackedLine.Estop :=
	        NOT (#cmp.PackedLine_Value0 = DB_Global.Status.Line.PackedLine.Estop);
	        
	        // Manual
	        // initial status: global MANUAL is deactivated
	        // If any of the conveyor gets MANUAL status; global MANUAL -> activated
	        #Line.PackedLine.Manual :=
	        NOT (#cmp.PackedLine_Value0 = DB_Global.Status.Line.PackedLine.Manual);
	        
	        // stop
	        // initial status: global STOP is deactivated
	        // If any of the conveyor gets STOP status; global stop -> activated
	        #Line.PackedLine.Stop :=
	        NOT (#cmp.PackedLine_Value0 = DB_Global.Status.Line.PackedLine.Stop);
	        
	    END_REGION
	    
	    REGION Line EmptyLine color for HMI
	        
	        // each and every status of the conveyor will be mentioned by different colors in HMI panel
	        
	        #ForVisu.Line.PackedLine.%X8 := #Line.PackedLine.Blockage;
	        // for future
	        (* OR
	        "IDB_KeyenceBP-I".TriggerSensorBlocked OR
	        "IDB_HeightSensor".BlockageActive *)
	        #ForVisu.Line.PackedLine.%X0 := #Line.PackedLine.ON;
	        #ForVisu.Line.PackedLine.%X1 := #Line.PackedLine.ReadytoRun;
	        #ForVisu.Line.PackedLine.%X2 := #Line.PackedLine.Occupied;
	        #ForVisu.Line.PackedLine.%X3 := #Line.PackedLine.Running;
	        #ForVisu.Line.PackedLine.%X4 := #Line.PackedLine.Fault;
	        #ForVisu.Line.PackedLine.%X5 := #Line.PackedLine.Estop;
	        #ForVisu.Line.PackedLine.%X6 := #Line.PackedLine.Manual;
	        #ForVisu.Line.PackedLine.%X7 := #Line.PackedLine.Stop;
	        
	        // convert word to Interger value: 
	        // color will be depends on the status priority (integer value) 
	        // reference: Conveyor image in HMI screen -> property -> Apperance   
	        
	        DB_VisuColor.Line.PackedLine.GlobalStatus :=
	        WORD_TO_INT(#ForVisu.Line.PackedLine);
	        
	    END_REGION
	    
	END_REGION
END_FUNCTION_BLOCK
END_NAMESPACE

NAMESPACE Global
ORGANIZATION_BLOCK Main_Global
TITLE = "Main Program Sweep (Cycle)"
{ S7_Optimized_Access := 'TRUE' ; Published := 'FALSE' }
VERSION : 0.1

BEGIN
	// ===
	// GoW
	// ==========================================================================================================================================
	// Company        : LogTech, s.r.o.
	// Created by     : Mahmoud Elnady
	// Block          : Main_Global
	// Project        : Lékarna DC Chrudim
	// Project number : 23-157
	// ==========================================================================================================================================
	
	REGION Global Status
	    
	    // All conveyor status
	    // For monitoring the whole system in simple way
	    // Global status is used for Klaxon lamp
	    IDB_GlobalStatus();
	    
	END_REGION
	
	REGION System
	    
	    FC_ReadSystemSSR();
	    
	END_REGION
	
	REGION MANUAL CONTROL
	    
	    IDB_ManualControl();
	    
	END_REGION
	
	
	REGION Hardware diag
	    
	    IDB_HardwareDiag();
	    
	END_REGION
	
	REGION HMI
	    
	    FC_SafetyAlarm();
	    
	    IDB_VisuAlarm();
	    
	END_REGION
	
	
	REGION Klaxon
	    
	    FC_AllKlaxon();
	    
	END_REGION
	
	
	
	
END_ORGANIZATION_BLOCK
END_NAMESPACE

NAMESPACE PackedLine
FUNCTION_BLOCK FB_PackedLine
{ S7_Optimized_Access := 'TRUE' ; Published := 'TRUE' }
VERSION : 0.1
   VAR 
      "G1.1.1" : _.Global.FB_Conveyor;
      "G1.1.2" : _.Global.FB_Conveyor;
      "G1.1.3" : _.Global.FB_Conveyor;
      "G1.1.4" : _.Global.FB_Conveyor;
      "G1.1.5" : _.Global.FB_Conveyor;
      "G1.1.6" : _.Global.FB_Conveyor;
      "G1.1.7" : _.Global.FB_Conveyor;
      "G1.1.8" : _.Global.FB_Conveyor;
      "G1.1.9" : _.Global.FB_Conveyor;
      "G1.1.10" : _.Global.FB_Conveyor;
      "G1.1.11" : _.Global.FB_Conveyor;
      "G1.1.12" : _.Global.FB_Conveyor;
      "G1.1.13" : _.Global.FB_Conveyor;
      "G1.1.14" : _.Global.FB_Conveyor;
      "G1.1.15" : _.Global.FB_Conveyor;
      "G1.1.16" : _.Global.FB_Conveyor;
      "G1.1.17" : _.Global.FB_Conveyor;
      "G1.1.18" : _.Global.FB_Conveyor;
      "G1.1.19" : _.Global.FB_Conveyor;
      "G1.2.1" : _.Global.FB_Conveyor;
      "G1.2.2" : _.Global.FB_Conveyor;
      "G1.3.1" : _.Global.FB_Conveyor;
      "G1.4.1" : _.Global.FB_Conveyor;
      "G1.4.2" : _.Global.FB_Conveyor;
      "G1.4.3" : _.Global.FB_Conveyor;
      "G1.4.4" : _.Global.FB_Conveyor;
      "G1.4.5" : _.Global.FB_Conveyor;
      "G1.4.6" : _.Global.FB_Conveyor;
      "G1.5.1" : _.Global.FB_Conveyor;
      "G1.5.2" : _.Global.FB_Conveyor;
      "G1.5.3" : _.Global.FB_Conveyor;
      "G1.5.4" : _.Global.FB_Conveyor;
      "G1.5.5" : _.Global.FB_Conveyor;
      "G1.5.6" : _.Global.FB_Conveyor;
      "G1.6.1" : _.Global.FB_Conveyor;
      "G1.6.2" : _.Global.FB_Conveyor;
      "G1.7.1" : _.Global.FB_Conveyor;
      "G1.7.2" : _.Global.FB_Conveyor;
      "G1.7.3" : _.Global.FB_Conveyor;
      "G1.7.4" : _.Global.FB_Conveyor;
   END_VAR


BEGIN
	// ==========================================================================================================================================
	// Company        : LogTech, s.r.o.
	// Created by     : Mahmoud Elnady
	// Block          : FB_Main_LineA1
	// Project        : Lékárna Chrudim
	// Project number : 23-157
	// ==========================================================================================================================================
	
	REGION G1.1.1
	    //G1.1.1
	    #"G1.1.1"(ConveyorID:=_."G1.1.1",
	              ConveyorSensor:=_."ASiGW-MCC001-bw200-C2: Input"."Sensor G1.1.1",
	                   Fault:= DB_UDI.PackedLine.Fault.Stop.Conveyor[_."G1.1.1"],
	                   Upstream:= DB_UDI.PackedLine.Upstream.Conveyor[_."G1.1.1"],
	                   Downstream:= DB_UDI.PackedLine.DownstreamAcu.Stop.Conveyor[_."G1.1.1"],
	                   Interlock:= DB_UDI.PackedLine.Interlock.Stop.Conveyor[_."G1.1.1"],
	                   RunForward=>_."ASiGW-MCC001-bw200-C2: Output"."Motor G1.1.1",
	                   WriteAsiDir=>_."ASiGW-MCC001-bw200-C2: Output"."Dir G1.1.1");
	         
	END_REGION
	
	REGION G1.1.2
	    //G1.1.2
	    #"G1.1.2"(ConveyorID := _."G1.1.2",
	              Fault := DB_UDI.PackedLine.Fault.Stop.Conveyor[_."G1.1.2"],
	              Upstream := DB_UDI.PackedLine.Upstream.Conveyor[_."G1.1.2"],
	              Downstream := DB_UDI.PackedLine.DownstreamAcu.Stop.Conveyor[_."G1.1.2"],
	              Interlock := DB_UDI.PackedLine.Interlock.Stop.Conveyor[_."G1.1.2"],
	              RunForward => _."ASiGW-MCC001-bw200-C2: Output"."Motor G1.1.2",
	              WriteAsiDir => _."ASiGW-MCC001-bw200-C2: Output"."Dir G1.1.2");
	    
	END_REGION
	
	REGION G1.1.3
	    //G1.1.3
	    #"G1.1.3"(ConveyorID := _."G1.1.3",
	              Fault := DB_UDI.PackedLine.Fault.Stop.Conveyor[_."G1.1.3"],
	              Upstream := DB_UDI.PackedLine.Upstream.Conveyor[_."G1.1.3"],
	              Downstream := DB_UDI.PackedLine.DownstreamAcu.Stop.Conveyor[_."G1.1.3"],
	              Interlock := DB_UDI.PackedLine.Interlock.Stop.Conveyor[_."G1.1.3"],
	              RunForward => _."ASiGW-MCC001-bw200-C2: Output"."Motor G1.1.3",
	              WriteAsiDir => _."ASiGW-MCC001-bw200-C2: Output"."Dir G1.1.3");
	    
	END_REGION
	
	REGION G1.1.4
	    //G1.1.4
	    #"G1.1.4"(ConveyorID:=_."G1.1.4",
	                   Fault:= DB_UDI.PackedLine.Fault.Stop.Conveyor[_."G1.1.4"],
	                   Upstream:= DB_UDI.PackedLine.Upstream.Conveyor[_."G1.1.4"],
	                   Downstream:= DB_UDI.PackedLine.DownstreamAcu.Stop.Conveyor[_."G1.1.4"],
	                   Interlock:= DB_UDI.PackedLine.Interlock.Stop.Conveyor[_."G1.1.4"],
	                   RunForward=>_."ASiGW-MCC001-bw200-C2: Output"."Motor G1.1.4",
	                   WriteAsiDir=>_."ASiGW-MCC001-bw200-C2: Output"."Dir G1.1.4");
	
	END_REGION
	
	REGION G1.1.5
	    //G1.1.5
	    #"G1.1.5"(ConveyorID:=_."G1.1.5",
	                   Fault:= DB_UDI.PackedLine.Fault.Stop.Conveyor[_."G1.1.5"],
	                   Upstream:= DB_UDI.PackedLine.Upstream.Conveyor[_."G1.1.5"],
	                   Downstream:= DB_UDI.PackedLine.DownstreamAcu.Stop.Conveyor[_."G1.1.5"],
	                   Interlock:= DB_UDI.PackedLine.Interlock.Stop.Conveyor[_."G1.1.5"],
	                   RunForward=>_."ASiGW-MCC001-bw200-C2: Output"."Motor G1.1.5",
	                   WriteAsiDir=>_."ASiGW-MCC001-bw200-C2: Output"."Dir G1.1.5");
	
	END_REGION
	
	REGION G1.1.6
	    //G1.1.6
	    #"G1.1.6"(ConveyorID:=_."G1.1.6",
	                   Fault:= DB_UDI.PackedLine.Fault.Stop.Conveyor[_."G1.1.6"],
	                   Upstream:= DB_UDI.PackedLine.Upstream.Conveyor[_."G1.1.6"],
	                   Downstream:= DB_UDI.PackedLine.DownstreamAcu.Stop.Conveyor[_."G1.1.6"],
	                   Interlock:= DB_UDI.PackedLine.Interlock.Stop.Conveyor[_."G1.1.6"],
	                   RunForward=>_."ASiGW-MCC001-bw200-C2: Output"."Motor G1.1.6",
	                   WriteAsiDir=>_."ASiGW-MCC001-bw200-C2: Output"."Dir G1.1.6");
	
	END_REGION
	
	REGION G1.1.7
	    //G1.1.7
	    #"G1.1.7"(ConveyorID := _."G1.1.7",
	              Fault := DB_UDI.PackedLine.Fault.Stop.Conveyor[_."G1.1.7"],
	              Upstream := DB_UDI.PackedLine.Upstream.Conveyor[_."G1.1.7"],
	              Downstream := DB_UDI.PackedLine.DownstreamAcu.Stop.Conveyor[_."G1.1.7"],
	              Interlock := DB_UDI.PackedLine.Interlock.Stop.Conveyor[_."G1.1.7"],
	              RunForward => _."ASiGW-MCC001-bw200-C2: Output"."Motor G1.1.7",
	              WriteAsiDir => _."ASiGW-MCC001-bw200-C2: Output"."Dir G1.1.7");
	    
	END_REGION
	
	REGION G1.1.8
	    //G1.1.8
	    #"G1.1.8"(ConveyorID := _."G1.1.8",
	              Fault := DB_UDI.PackedLine.Fault.Stop.Conveyor[_."G1.1.8"],
	              Upstream := DB_UDI.PackedLine.Upstream.Conveyor[_."G1.1.8"],
	              Downstream := DB_UDI.PackedLine.DownstreamAcu.Stop.Conveyor[_."G1.1.8"],
	              Interlock := DB_UDI.PackedLine.Interlock.Stop.Conveyor[_."G1.1.8"],
	              RunForward => _."ASiGW-MCC001-bw200-C2: Output"."Motor G1.1.8",
	              WriteAsiDir => _."ASiGW-MCC001-bw200-C2: Output"."Dir G1.1.8");
	    
	END_REGION
	
	REGION G1.1.9
	    //G1.1.9
	    #"G1.1.9"(ConveyorID:=_."G1.1.9",
	                   Fault:= DB_UDI.PackedLine.Fault.Stop.Conveyor[_."G1.1.9"],
	                   Upstream:= DB_UDI.PackedLine.Upstream.Conveyor[_."G1.1.9"],
	                   Downstream:= DB_UDI.PackedLine.DownstreamAcu.Stop.Conveyor[_."G1.1.9"],
	                   Interlock:= DB_UDI.PackedLine.Interlock.Stop.Conveyor[_."G1.1.9"],
	                   RunForward=>_."ASiGW-MCC001-bw200-C2: Output"."Motor G1.1.9",
	                   WriteAsiDir=>_."ASiGW-MCC001-bw200-C2: Output"."Dir G1.1.9");
	         
	END_REGION
	
	REGION G1.1.10
	    //G1.1.10
	    #"G1.1.10"(ConveyorID:=_."G1.1.10",
	               ConveyorSensor:=_."ASiGW-MCC001-bw200-C2: Input"."Sensor G1.1.10",
	                   Fault:= DB_UDI.PackedLine.Fault.Stop.Conveyor[_."G1.1.10"],
	                   Upstream:= DB_UDI.PackedLine.Upstream.Conveyor[_."G1.1.10"],
	                   Downstream:= DB_UDI.PackedLine.DownstreamAcu.Stop.Conveyor[_."G1.1.10"],
	                   Interlock:= DB_UDI.PackedLine.Interlock.Stop.Conveyor[_."G1.1.10"],
	                   RunForward=>_."ASiGW-MCC001-bw200-C2: Output"."Motor G1.1.10",
	                   WriteAsiDir=>_."ASiGW-MCC001-bw200-C2: Output"."Dir G1.1.10");
	
	END_REGION
	
	REGION G1.1.11
	    //G1.1.11
	    #"G1.1.11"(ConveyorID := _."G1.1.11",
	               Fault := DB_UDI.PackedLine.Fault.Stop.Conveyor[_."G1.1.11"],
	               Upstream := DB_UDI.PackedLine.Upstream.Conveyor[_."G1.1.11"],
	               Downstream := DB_UDI.PackedLine.DownstreamAcu.Stop.Conveyor[_."G1.1.11"],
	               Interlock := DB_UDI.PackedLine.Interlock.Stop.Conveyor[_."G1.1.11"],
	               RunForward => _."ASiGW-MCC001-bw200-C2: Output"."Motor G1.1.11",
	               WriteAsiDir => _."ASiGW-MCC001-bw200-C2: Output"."Dir G1.1.11");
	    
	END_REGION
	
	REGION G1.1.12
	    //G1.1.12
	    #"G1.1.12"(ConveyorID:=_."G1.1.12",
	                   Fault:= DB_UDI.PackedLine.Fault.Stop.Conveyor[_."G1.1.12"],
	                   Upstream:= DB_UDI.PackedLine.Upstream.Conveyor[_."G1.1.12"],
	                   Downstream:= DB_UDI.PackedLine.DownstreamAcu.Stop.Conveyor[_."G1.1.12"],
	                   Interlock:= DB_UDI.PackedLine.Interlock.Stop.Conveyor[_."G1.1.12"],
	                   RunForward=>_."ASiGW-MCC001-bw200-C2: Output"."Motor G1.1.12",
	                   WriteAsiDir=>_."ASiGW-MCC001-bw200-C2: Output"."Dir G1.1.12");
	
	END_REGION
	
	REGION G1.1.13
	    //G1.1.13
	    #"G1.1.13"(ConveyorID:=_."G1.1.13",
	                   Fault:= DB_UDI.PackedLine.Fault.Stop.Conveyor[_."G1.1.13"],
	                   Upstream:= DB_UDI.PackedLine.Upstream.Conveyor[_."G1.1.13"],
	                   Downstream:= DB_UDI.PackedLine.DownstreamAcu.Stop.Conveyor[_."G1.1.13"],
	                   Interlock:= DB_UDI.PackedLine.Interlock.Stop.Conveyor[_."G1.1.13"],
	                   RunForward=>_."ASiGW-MCC001-bw200-C2: Output"."Motor G1.1.13",
	                   WriteAsiDir=>_."ASiGW-MCC001-bw200-C2: Output"."Dir G1.1.13");
	
	END_REGION
	
	REGION G1.1.14
	    //G1.1.14
	    #"G1.1.14"(ConveyorID:=_."G1.1.14",
	                   Fault:= DB_UDI.PackedLine.Fault.Stop.Conveyor[_."G1.1.14"],
	                   Upstream:= DB_UDI.PackedLine.Upstream.Conveyor[_."G1.1.14"],
	                   Downstream:= DB_UDI.PackedLine.DownstreamAcu.Stop.Conveyor[_."G1.1.14"],
	                   Interlock:= DB_UDI.PackedLine.Interlock.Stop.Conveyor[_."G1.1.14"],
	                   RunForward=>_."ASiGW-MCC001-bw200-C2: Output"."Motor G1.1.14",
	                   WriteAsiDir=>_."ASiGW-MCC001-bw200-C2: Output"."Dir G1.1.14");
	
	END_REGION
	
	REGION G1.1.15
	    //G1.1.15
	    #"G1.1.15"(ConveyorID:=_."G1.1.15",
	                   Fault:= DB_UDI.PackedLine.Fault.Stop.Conveyor[_."G1.1.15"],
	                   Upstream:= DB_UDI.PackedLine.Upstream.Conveyor[_."G1.1.15"],
	                   Downstream:= DB_UDI.PackedLine.DownstreamAcu.Stop.Conveyor[_."G1.1.15"],
	                   Interlock:= DB_UDI.PackedLine.Interlock.Stop.Conveyor[_."G1.1.15"],
	                   RunForward=>_."ASiGW-MCC001-bw200-C2: Output"."Motor G1.1.15",
	                   WriteAsiDir=>_."ASiGW-MCC001-bw200-C2: Output"."Dir G1.1.15");
	
	END_REGION
	
	REGION G1.1.16
	    //G1.1.16
	    #"G1.1.16"(ConveyorID:=_."G1.1.16",
	                   Fault:= DB_UDI.PackedLine.Fault.Stop.Conveyor[_."G1.1.16"],
	                   Upstream:= DB_UDI.PackedLine.Upstream.Conveyor[_."G1.1.16"],
	                   Downstream:= DB_UDI.PackedLine.DownstreamAcu.Stop.Conveyor[_."G1.1.16"],
	                   Interlock:= DB_UDI.PackedLine.Interlock.Stop.Conveyor[_."G1.1.16"],
	                   RunForward=>_."ASiGW-MCC001-bw200-C2: Output"."Motor G1.1.16",
	                   WriteAsiDir=>_."ASiGW-MCC001-bw200-C2: Output"."Dir G1.1.16");
	        
	END_REGION
	
	REGION G1.1.17
	    //G1.1.17
	    #"G1.1.17"(ConveyorID := _."G1.1.17",
	               Fault := DB_UDI.PackedLine.Fault.Stop.Conveyor[_."G1.1.17"],
	               Upstream := DB_UDI.PackedLine.Upstream.Conveyor[_."G1.1.17"],
	               Downstream := DB_UDI.PackedLine.DownstreamAcu.Stop.Conveyor[_."G1.1.17"],
	               Interlock := DB_UDI.PackedLine.Interlock.Stop.Conveyor[_."G1.1.17"],
	               RunForward => _."ASiGW-MCC001-bw200-C2: Output"."Motor G1.1.17",
	               WriteAsiDir => _."ASiGW-MCC001-bw200-C2: Output"."Dir G1.1.17");
	
	END_REGION
	
	REGION G1.1.18
	    //G1.1.18
	    #"G1.1.18"(ConveyorID:=_."G1.1.18",
	                   Fault:= DB_UDI.PackedLine.Fault.Stop.Conveyor[_."G1.1.18"],
	                   Upstream:= DB_UDI.PackedLine.Upstream.Conveyor[_."G1.1.18"],
	                   Downstream:= DB_UDI.PackedLine.DownstreamAcu.Stop.Conveyor[_."G1.1.18"],
	                   Interlock:= DB_UDI.PackedLine.Interlock.Stop.Conveyor[_."G1.1.18"],
	                   RunForward=>_."ASiGW-MCC001-bw200-C2: Output"."Motor G1.1.18",
	                   WriteAsiDir=>_."ASiGW-MCC001-bw200-C2: Output"."Dir G1.1.18");
	        
	END_REGION
	
	REGION G1.1.19
	    //G1.1.19
	    #"G1.1.19"(ConveyorID:=_."G1.1.19",
	               ConveyorSensor:=_."ASiGW-MCC001-bw200-C2: Input"."Sensor G1.1.19",
	                   Fault:= DB_UDI.PackedLine.Fault.Stop.Conveyor[_."G1.1.19"],
	                   Upstream:= DB_UDI.PackedLine.Upstream.Conveyor[_."G1.1.19"],
	                   Downstream:= DB_UDI.PackedLine.DownstreamAcu.Stop.Conveyor[_."G1.1.19"],
	                   Interlock:= DB_UDI.PackedLine.Interlock.Stop.Conveyor[_."G1.1.19"],
	                   RunForward=>_."ASiGW-MCC001-bw200-C2: Output"."Motor G1.1.19",
	                   WriteAsiDir=>_."ASiGW-MCC001-bw200-C2: Output"."Dir G1.1.19");
	        
	END_REGION
	
	REGION G1.2.1
	    //G1.2.1
	    #"G1.2.1"(ConveyorID := _."G1.2.1",
	              ConveyorSensor:=_."ASiGW-MCC001-bw200-C2: Input"."Sensor G1.2.1",
	              Fault := DB_UDI.PackedLine.Fault.Stop.Conveyor[_."G1.2.1"],
	              Upstream := DB_UDI.PackedLine.Upstream.Conveyor[_."G1.2.1"],
	              Downstream := DB_UDI.PackedLine.DownstreamAcu.Stop.Conveyor[_."G1.2.1"],
	              Interlock := DB_UDI.PackedLine.Interlock.Stop.Conveyor[_."G1.2.1"],
	              RunForward => _."ASiGW-MCC001-bw200-C2: Output"."Motor - G1.2.1",
	              WriteAsiDir => _."ASiGW-MCC001-bw200-C2: Output"."2-11B Dir",
	              WriteAsiSpeed=> _."ASiGW-MCC001-bw200-C2: Output"."2-11B Speed");
	    
	END_REGION
	
	REGION G1.2.2
	    //G1.2.2
	    #"G1.2.2"(ConveyorID:=_."G1.2.2",
	              ConveyorSensor:=_."ASiGW-MCC001-bw200-C2: Input"."Sensor G1.2.2",
	                   Fault:= DB_UDI.PackedLine.Fault.Stop.Conveyor[_."G1.2.2"],
	                   Upstream:= DB_UDI.PackedLine.Upstream.Conveyor[_."G1.2.2"],
	                   Downstream:= DB_UDI.PackedLine.DownstreamAcu.Stop.Conveyor[_."G1.2.2"],
	                   Interlock:= DB_UDI.PackedLine.Interlock.Stop.Conveyor[_."G1.2.2"],
	                   RunForward => _."ASiGW-MCC001-bw200-C2: Output"."Motor - G1.2.2",
	                   WriteAsiDir => _."ASiGW-MCC001-bw200-C2: Output"."2-11B Dir",
	                   WriteAsiSpeed=> _."ASiGW-MCC001-bw200-C2: Output"."2-11B Speed");
	
	END_REGION
	
	REGION G1.3.1
	    //G1.3.1
	    #"G1.3.1"(ConveyorID:=_."G1.3.1",
	                   Fault:= DB_UDI.PackedLine.Fault.Stop.Conveyor[_."G1.3.1"],
	                   Upstream:= DB_UDI.PackedLine.Upstream.Conveyor[_."G1.3.1"],
	                   Downstream:= DB_UDI.PackedLine.DownstreamAcu.Stop.Conveyor[_."G1.3.1"],
	                   Interlock:= DB_UDI.PackedLine.Interlock.Stop.Conveyor[_."G1.3.1"],
	                   ImcSpeed=>_."IMC84MotorTargetSpeedRD -G1.3.1");
	END_REGION
	
	REGION G1.4.1
	    //G1.4.1
	    #"G1.4.1"(ConveyorID:=_."G1.4.1",
	                   Fault:= DB_UDI.PackedLine.Fault.Stop.Conveyor[_."G1.4.1"],
	                   Upstream:= DB_UDI.PackedLine.Upstream.Conveyor[_."G1.4.1"],
	                   Downstream:= DB_UDI.PackedLine.DownstreamAcu.Stop.Conveyor[_."G1.4.1"],
	                   Interlock:= DB_UDI.PackedLine.Interlock.Stop.Conveyor[_."G1.4.1"],
	                   ImcSpeed=>_."IMC84MotorTargetSpeedRD -G1.4.1");
	
	END_REGION
	
	REGION G1.4.2
	    //G1.4.2
	    #"G1.4.2"(ConveyorID:=_."G1.4.2",
	                   Fault:= DB_UDI.PackedLine.Fault.Stop.Conveyor[_."G1.4.2"],
	                   Upstream:= DB_UDI.PackedLine.Upstream.Conveyor[_."G1.4.2"],
	                   Downstream:= DB_UDI.PackedLine.DownstreamAcu.Stop.Conveyor[_."G1.4.2"],
	                   Interlock:= DB_UDI.PackedLine.Interlock.Stop.Conveyor[_."G1.4.2"],
	                   ImcSpeed=>_."IMC84MotorTargetSpeedRD -G1.4.2");
	
	END_REGION
	
	REGION G1.4.3
	    //G1.4.3
	    #"G1.4.3"(ConveyorID := _."G1.4.3",
	              Fault := DB_UDI.PackedLine.Fault.Stop.Conveyor[_."G1.4.3"],
	              Upstream := DB_UDI.PackedLine.Upstream.Conveyor[_."G1.4.3"],
	              Downstream := DB_UDI.PackedLine.DownstreamAcu.Stop.Conveyor[_."G1.4.3"],
	              Interlock := DB_UDI.PackedLine.Interlock.Stop.Conveyor[_."G1.4.3"],
	              ImcSpeed=>_."IMC84MotorTargetSpeedRD -G1.4.3");
	    
	END_REGION
	
	REGION G1.4.4
	    //G1.4.4
	    #"G1.4.4"(ConveyorID := _."G1.4.4",
	              Fault := DB_UDI.PackedLine.Fault.Stop.Conveyor[_."G1.4.4"],
	              Upstream := DB_UDI.PackedLine.Upstream.Conveyor[_."G1.4.4"],
	              Downstream := DB_UDI.PackedLine.DownstreamAcu.Stop.Conveyor[_."G1.4.4"],
	              Interlock := DB_UDI.PackedLine.Interlock.Stop.Conveyor[_."G1.4.4"],
	              ImcSpeed => _."IMC85MotorTargetSpeedRD -G1.4.4");
	    
	END_REGION
	
	REGION G1.4.5
	    //G1.4.5
	    #"G1.4.5"(ConveyorID:=_."G1.4.5",
	                   Fault:= DB_UDI.PackedLine.Fault.Stop.Conveyor[_."G1.4.5"],
	                   Upstream:= DB_UDI.PackedLine.Upstream.Conveyor[_."G1.4.5"],
	                   Downstream:= DB_UDI.PackedLine.DownstreamAcu.Stop.Conveyor[_."G1.4.5"],
	                   Interlock:= DB_UDI.PackedLine.Interlock.Stop.Conveyor[_."G1.4.5"],
	                   ImcSpeed=>_."IMC85MotorTargetSpeedRD -G1.4.5");
	
	END_REGION
	
	REGION G1.4.6
	    //G1.4.6
	    #"G1.4.6"(ConveyorID := _."G1.4.6",
	              Fault := DB_UDI.PackedLine.Fault.Stop.Conveyor[_."G1.4.6"],
	              Upstream := DB_UDI.PackedLine.Upstream.Conveyor[_."G1.4.6"],
	              Downstream := DB_UDI.PackedLine.DownstreamAcu.Stop.Conveyor[_."G1.4.6"],
	              Interlock := DB_UDI.PackedLine.Interlock.Stop.Conveyor[_."G1.4.6"],
	              ImcSpeed => _."IMC85MotorTargetSpeedRD -G1.4.6");
	    
	END_REGION
	
	REGION G1.5.1
	    //G1.5.1
	    #"G1.5.1"(ConveyorID := _."G1.5.1",
	              Fault := DB_UDI.PackedLine.Fault.Stop.Conveyor[_."G1.5.1"],
	              Upstream := DB_UDI.PackedLine.Upstream.Conveyor[_."G1.5.1"],
	              Downstream := DB_UDI.PackedLine.DownstreamAcu.Stop.Conveyor[_."G1.5.1"],
	              Interlock := DB_UDI.PackedLine.Interlock.Stop.Conveyor[_."G1.5.1"],
	              ImcSpeed => _."IMC85MotorTargetSpeedRD -G1.5.1");
	    
	END_REGION
	
	REGION G1.5.2
	    //G1.5.2
	    #"G1.5.2"(ConveyorID := _."G1.5.2",
	              Fault := DB_UDI.PackedLine.Fault.Stop.Conveyor[_."G1.5.2"],
	              Upstream := DB_UDI.PackedLine.Upstream.Conveyor[_."G1.5.2"],
	              Downstream := DB_UDI.PackedLine.DownstreamAcu.Stop.Conveyor[_."G1.5.2"],
	              Interlock := DB_UDI.PackedLine.Interlock.Stop.Conveyor[_."G1.5.2"],
	              ImcSpeed => _."IMC86MotorTargetSpeedRD -G1.5.2");
	    
	END_REGION
	
	REGION G1.5.3
	    //G1.5.3
	    #"G1.5.3"(ConveyorID := _."G1.5.3",
	              Fault := DB_UDI.PackedLine.Fault.Stop.Conveyor[_."G1.5.3"],
	              Upstream := DB_UDI.PackedLine.Upstream.Conveyor[_."G1.5.3"],
	              Downstream := DB_UDI.PackedLine.DownstreamAcu.Stop.Conveyor[_."G1.5.3"],
	              Interlock := DB_UDI.PackedLine.Interlock.Stop.Conveyor[_."G1.5.3"],
	              ImcSpeed => _."IMC86MotorTargetSpeedRD -G1.5.3");
	    
	END_REGION
	
	REGION G1.5.4
	    //G1.5.4
	    #"G1.5.4"(ConveyorID := _."G1.5.4",
	              Fault := DB_UDI.PackedLine.Fault.Stop.Conveyor[_."G1.5.4"],
	              Upstream := DB_UDI.PackedLine.Upstream.Conveyor[_."G1.5.4"],
	              Downstream := DB_UDI.PackedLine.DownstreamAcu.Stop.Conveyor[_."G1.5.4"],
	              Interlock := DB_UDI.PackedLine.Interlock.Stop.Conveyor[_."G1.5.4"],
	              ImcSpeed=>_."IMC86MotorTargetSpeedRD -G1.5.4");
	    
	END_REGION
	
	REGION G1.5.5
	    //G1.5.5
	    #"G1.5.5"(ConveyorID:=_."G1.5.5",
	                   Fault:= DB_UDI.PackedLine.Fault.Stop.Conveyor[_."G1.5.5"],
	                   Upstream:= DB_UDI.PackedLine.Upstream.Conveyor[_."G1.5.5"],
	                   Downstream:= DB_UDI.PackedLine.DownstreamAcu.Stop.Conveyor[_."G1.5.5"],
	                   Interlock:= DB_UDI.PackedLine.Interlock.Stop.Conveyor[_."G1.5.5"],
	                   ImcSpeed=>_."IMC86MotorTargetSpeedRD -G1.5.5");
	         
	END_REGION
	
	REGION G1.5.6
	    //G1.5.6
	    #"G1.5.6"(ConveyorID := _."G1.5.6",
	              Fault := DB_UDI.PackedLine.Fault.Stop.Conveyor[_."G1.5.6"],
	              Upstream := DB_UDI.PackedLine.Upstream.Conveyor[_."G1.5.6"],
	              Downstream := DB_UDI.PackedLine.DownstreamAcu.Stop.Conveyor[_."G1.5.6"],
	              Interlock := DB_UDI.PackedLine.Interlock.Stop.Conveyor[_."G1.5.6"],
	              ImcSpeed => _."IMC87MotorTargetSpeedRD -G1.5.6");
	    
	END_REGION
	
	REGION G1.6.1
	    //G1.6.1
	    #"G1.6.1"(ConveyorID := _."G1.6.1",
	              ConveyorSensor := _."IMC84Sensor_2",
	              Fault := DB_UDI.PackedLine.Fault.Stop.Conveyor[_."G1.6.1"],
	              Upstream := DB_UDI.PackedLine.Upstream.Conveyor[_."G1.6.1"],
	              Downstream := DB_UDI.PackedLine.DownstreamAcu.Stop.Conveyor[_."G1.6.1"],
	              Interlock := DB_UDI.PackedLine.Interlock.Stop.Conveyor[_."G1.6.1"],
	              ImcSpeed => _."IMC87MotorTargetSpeedRD -G1.6.1");
	    
	END_REGION
	
	REGION G1.6.2
	    //G1.6.2
	    #"G1.6.2"(ConveyorID := _."G1.6.2",
	              ConveyorSensor := _."IMC84Sensor_3",
	              Fault := DB_UDI.PackedLine.Fault.Stop.Conveyor[_."G1.6.2"],
	              Upstream := DB_UDI.PackedLine.Upstream.Conveyor[_."G1.6.2"],
	              Downstream := DB_UDI.PackedLine.DownstreamAcu.Stop.Conveyor[_."G1.6.2"],
	              Interlock := DB_UDI.PackedLine.Interlock.Stop.Conveyor[_."G1.6.2"],
	              ImcSpeed => _."IMC87MotorTargetSpeedRD -G1.6.2");
	    
	END_REGION
	
	REGION G1.7.1
	    //G1.7.1
	    #"G1.7.1"(ConveyorID:=_."G1.7.1",
	                   Fault:= DB_UDI.PackedLine.Fault.Stop.Conveyor[_."G1.7.1"],
	                   Upstream:= DB_UDI.PackedLine.Upstream.Conveyor[_."G1.7.1"],
	                   Downstream:= DB_UDI.PackedLine.DownstreamAcu.Stop.Conveyor[_."G1.7.1"],
	                   Interlock:= DB_UDI.PackedLine.Interlock.Stop.Conveyor[_."G1.7.1"],
	                   ImcSpeed=>_."IMC87MotorTargetSpeedRD -G1.7.1");
	
	END_REGION
	
	REGION G1.7.2
	    //G1.7.2
	    #"G1.7.2"(ConveyorID:=_."G1.7.2",
	                   Fault:= DB_UDI.PackedLine.Fault.Stop.Conveyor[_."G1.7.2"],
	                   Upstream:= DB_UDI.PackedLine.Upstream.Conveyor[_."G1.7.2"],
	                   Downstream:= DB_UDI.PackedLine.DownstreamAcu.Stop.Conveyor[_."G1.7.2"],
	                   Interlock:= DB_UDI.PackedLine.Interlock.Stop.Conveyor[_."G1.7.2"],
	                   ImcSpeed=>_."IMC88MotorTargetSpeedRD -G1.7.2");
	
	END_REGION
	
	REGION G1.7.3
	    //G1.7.3
	    #"G1.7.3"(ConveyorID := _."G1.7.3",
	              Fault := DB_UDI.PackedLine.Fault.Stop.Conveyor[_."G1.7.3"],
	              Upstream := DB_UDI.PackedLine.Upstream.Conveyor[_."G1.7.3"],
	              Downstream := DB_UDI.PackedLine.DownstreamAcu.Stop.Conveyor[_."G1.7.3"],
	              Interlock := DB_UDI.PackedLine.Interlock.Stop.Conveyor[_."G1.7.3"],
	              ImcSpeed=>_."IMC88MotorTargetSpeedRD -G1.7.3");
	    
	END_REGION
	
	REGION G1.7.4
	    //G1.7.4
	    #"G1.7.4"(ConveyorID := _."G1.7.4",
	              ConveyorSensor := _."IMC88Sensor_4",
	              Fault := DB_UDI.PackedLine.Fault.Stop.Conveyor[_."G1.7.4"],
	              Upstream := DB_UDI.PackedLine.Upstream.Conveyor[_."G1.7.4"],
	              Downstream := DB_UDI.PackedLine.DownstreamAcu.Stop.Conveyor[_."G1.7.4"],
	              Interlock := DB_UDI.PackedLine.Interlock.Stop.Conveyor[_."G1.7.4"],
	              ImcSpeed => _."IMC88MotorTargetSpeedRD -G1.7.4");
	    
	END_REGION
	
	
	
	
	
	
	
	
	
	
	
	
	
	
	
	
END_FUNCTION_BLOCK
END_NAMESPACE

NAMESPACE PackedLine
ORGANIZATION_BLOCK Main_PackedLine
TITLE = "Main Program Sweep (Cycle)"
{ S7_Optimized_Access := 'TRUE' ; Published := 'FALSE' }
VERSION : 0.1

BEGIN
	IDB_PackedLine();
	
END_ORGANIZATION_BLOCK
END_NAMESPACE

NAMESPACE ProductionLine
ORGANIZATION_BLOCK CyclicInterrupt
{ S7_Optimized_Access := 'TRUE' ; Published := 'FALSE' }
VERSION : 0.1

BEGIN
	// ==========================================================================================================================================
	// Company        : LogTech, s.r.o.
	// Created by     : Mahmoud Elnady
	// Block          : CyclicInterrupt
	// Project        : Lékarna DC Chrudim
	// Project number : 23-157
	// ==========================================================================================================================================
	
	REGION B1.6.1 Transfer Unit
	    
	    IDB_S300_FullControl(TransferID:=_."B1.6.1",
	                         TransferSensor:=_."ASiGW-MCC001-bw143-C1: Input"."LoadPresence -B1.6.1",
	                         RollerUp:= _."ASiGW-MCC001-bw143-C1: Input"."Up/Down -B1.6.1",
	                         Fault:=DB_UDI.ProductionLine.Fault.Stop.Conveyor[_."B1.6.1"],
	                         ReadyToRCV:=DB_UDI.ProductionLine.Fault.Stop.Conveyor[_."B1.6.1"],
	                         UpstreamStraight:=IDB_ProductionLine."B1.5.1".FilteredSensor,
	                         UpstreamArm:=IDB_ProductionLine."B1.18.1".FilteredSensor,
	                         FrontSensor:= _."ASiGW-MCC001-bw143-C1: Input"."FrontSensor -B1.6.1",
	                         EndSensor:= _."ASiGW-MCC001-bw143-C1: Input"."EndSensor -B1.6.1",
	                         "Left/RightSensor":=_."ASiGW-MCC001-bw143-C1: Input"."LeftSensor -B1.6.1",
	                         Downstream:=DB_UDI.ProductionLine.DownstreamAccu.Stop.Conveyor[_."B1.6.1"],
	                         PriorityStraight:= IDB_Merging."Merge_B1.6.1".Priority.Straight,
	                         PriorityArm:= IDB_Merging."Merge_B1.6.1".Priority.Arm,
	                         Direction=> _."ASiGW-MCC001-bw143-C1: Output"."Direction -B1.6.1",
	                         Cmd1=>_."ASiGW-MCC001-bw143-C1: Output"."Command1 -B1.6.1",
	                         Cmd2=>_."ASiGW-MCC001-bw143-C1: Output"."Command2 -B1.6.1",
	                         ErrorReset=>_."ASiGW-MCC001-bw143-C1: Output"."ErrorReset -B1.6.1");
	    
	    
	END_REGION
	
	//IDB_ProductionLine."B1.6.1".ReadTransferStatus := IDB_S300_FullControl.ReadTransferStatus;
	
	//IDB_ProductionLine."B1.6.1".VisuColor := IDB_ProductionLine."B1.6.1".VisuColor;
	
	
END_ORGANIZATION_BLOCK
END_NAMESPACE

NAMESPACE ProductionLine
FUNCTION_BLOCK FB_ProductionLine
{ S7_Optimized_Access := 'TRUE' ; Published := 'TRUE' }
VERSION : 0.1
   VAR 
      "A1.1.1" : _.Global.FB_Conveyor;
      "A1.1.2" : _.Global.FB_Conveyor;
      "A1.1.3" : _.Global.FB_Conveyor;
      "A1.1.4" : _.Global.FB_Conveyor;
      "A1.1.5" : _.Global.FB_Conveyor;
      "A1.1.6" : _.Global.FB_Conveyor;
      "A1.1.7" : _.Global.FB_Conveyor;
      "A1.1.8" : _.Global.FB_Conveyor;
      "A1.1.9" : _.Global.FB_Conveyor;
      "A1.1.10" : _.Global.FB_Conveyor;
      "A1.1.11" : _.Global.FB_Conveyor;
      "A1.1.12" : _.Global.FB_Conveyor;
      "A1.1.13" : _.Global.FB_Conveyor;
      "A1.1.14" : _.Global.FB_Conveyor;
      "A1.2.1" : _.Global.FB_Conveyor;
      "A1.3.1" : _.Global.FB_Conveyor;
      "A1.4.1" : _.Global.FB_Conveyor;
      "A1.5.1" : _.Global.FB_Conveyor;
      "A1.5.2" : _.Global.FB_Conveyor;
      "A1.5.3" : _.Global.FB_Conveyor;
      "A1.7.1" : _.Global.FB_Conveyor;
      "A1.7.2" : _.Global.FB_Conveyor;
      "A1.7.3" : _.Global.FB_Conveyor;
      "A1.7.4" : _.Global.FB_Conveyor;
      "A1.7.5" : _.Global.FB_Conveyor;
      "A1.7.6" : _.Global.FB_Conveyor;
      "A1.8.1" : _.Global.FB_Conveyor;
      "A1.10.1" : _.Global.FB_Conveyor;
      "A1.10.2" : _.Global.FB_Conveyor;
      "A1.10.3" : _.Global.FB_Conveyor;
      "A1.10.4" : _.Global.FB_Conveyor;
      "A1.10.5" : _.Global.FB_Conveyor;
      "A1.10.6" : _.Global.FB_Conveyor;
      "A1.10.7" : _.Global.FB_Conveyor;
      "A1.10.8" : _.Global.FB_Conveyor;
      "A1.10.9" : _.Global.FB_Conveyor;
      "A1.10.10" : _.Global.FB_Conveyor;
      "A1.10.11" : _.Global.FB_Conveyor;
      "A1.10.12" : _.Global.FB_Conveyor;
      "A1.10.13" : _.Global.FB_Conveyor;
      "A1.11.1" : _.Global.FB_Conveyor;
      "A1.11.2" : _.Global.FB_Conveyor;
      "A1.12.1" : _.Global.FB_Conveyor;
      "A1.12.2" : _.Global.FB_Conveyor;
      "A1.14.1" : _.Global.FB_Conveyor;
      "A1.14.2" : _.Global.FB_Conveyor;
      "A1.14.3" : _.Global.FB_Conveyor;
      "A1.14.4" : _.Global.FB_Conveyor;
      "A1.14.5" : _.Global.FB_Conveyor;
      "A1.14.6" : _.Global.FB_Conveyor;
      "A1.14.7" : _.Global.FB_Conveyor;
      "A1.14.8" : _.Global.FB_Conveyor;
      "A1.14.9" : _.Global.FB_Conveyor;
      "A1.14.10" : _.Global.FB_Conveyor;
      "A1.14.11" : _.Global.FB_Conveyor;
      "A1.14.12" : _.Global.FB_Conveyor;
      "A1.14.13" : _.Global.FB_Conveyor;
      "A1.14.14" : _.Global.FB_Conveyor;
      "A1.14.15" : _.Global.FB_Conveyor;
      "A1.14.16" : _.Global.FB_Conveyor;
      "A1.14.17" : _.Global.FB_Conveyor;
      "A1.14.18" : _.Global.FB_Conveyor;
      "A1.14.19" : _.Global.FB_Conveyor;
      "A1.14.20" : _.Global.FB_Conveyor;
      "A1.14.21" : _.Global.FB_Conveyor;
      "A1.14.22" : _.Global.FB_Conveyor;
      "A1.14.23" : _.Global.FB_Conveyor;
      "A1.14.24" : _.Global.FB_Conveyor;
      "A1.14.25" : _.Global.FB_Conveyor;
      "A1.14.26" : _.Global.FB_Conveyor;
      "A2.2.1" : _.Global.FB_Conveyor;
      "A2.2.2" : _.Global.FB_Conveyor;
      "A2.2.3" : _.Global.FB_Conveyor;
      "A2.2.4" : _.Global.FB_Conveyor;
      "A2.2.5" : _.Global.FB_Conveyor;
      "A2.2.6" : _.Global.FB_Conveyor;
      "A2.2.7" : _.Global.FB_Conveyor;
      "A2.2.8" : _.Global.FB_Conveyor;
      "A2.2.9" : _.Global.FB_Conveyor;
      "A2.2.10" : _.Global.FB_Conveyor;
      "A2.2.11" : _.Global.FB_Conveyor;
      "A2.2.12" : _.Global.FB_Conveyor;
      "A2.2.13" : _.Global.FB_Conveyor;
      "A2.2.14" : _.Global.FB_Conveyor;
      "A2.2.15" : _.Global.FB_Conveyor;
      "A2.2.16" : _.Global.FB_Conveyor;
      "A2.2.17" : _.Global.FB_Conveyor;
      "A2.2.18" : _.Global.FB_Conveyor;
      "A2.2.19" : _.Global.FB_Conveyor;
      "A2.2.20" : _.Global.FB_Conveyor;
      "A2.2.21" : _.Global.FB_Conveyor;
      "A2.2.22" : _.Global.FB_Conveyor;
      "A2.2.23" : _.Global.FB_Conveyor;
      "A2.2.24" : _.Global.FB_Conveyor;
      "A2.2.25" : _.Global.FB_Conveyor;
      "A2.2.26" : _.Global.FB_Conveyor;
      "B1.1.1" : _.Global.FB_Conveyor;
      "B1.2.1" : _.Global.FB_Conveyor;
      "B1.3.1" : _.Global.FB_Conveyor;
      "B1.3.2" : _.Global.FB_Conveyor;
      "B1.3.3" : _.Global.FB_Conveyor;
      "B1.4.1" : _.Global.FB_Conveyor;
      "B1.4.2" : _.Global.FB_Conveyor;
      "B1.5.1" : _.Global.FB_Conveyor;
      "B1.7.1" : _.Global.FB_Conveyor;
      "B1.7.2" : _.Global.FB_Conveyor;
      "B1.7.3" : _.Global.FB_Conveyor;
      "B1.8.1" : _.Global.FB_Conveyor;
      "B1.8.2" : _.Global.FB_Conveyor;
      "B1.8.3" : _.Global.FB_Conveyor;
      "B1.9.1" : _.Global.FB_Conveyor;
      "B1.9.2" : _.Global.FB_Conveyor;
      "B1.11.1" : _.Global.FB_Conveyor;
      "B1.11.2" : _.Global.FB_Conveyor;
      "B1.11.3" : _.Global.FB_Conveyor;
      "B1.11.4" : _.Global.FB_Conveyor;
      "B1.12.1" : _.Global.FB_Conveyor;
      "B1.12.2" : _.Global.FB_Conveyor;
      "B1.15.1" : _.Global.FB_Conveyor;
      "B1.15.2" : _.Global.FB_Conveyor;
      "B1.16.1" : _.Global.FB_Conveyor;
      "B1.16.2" : _.Global.FB_Conveyor;
      "B1.16.3" : _.Global.FB_Conveyor;
      "B1.16.4" : _.Global.FB_Conveyor;
      "B1.16.5" : _.Global.FB_Conveyor;
      "B1.16.6" : _.Global.FB_Conveyor;
      "B1.16.7" : _.Global.FB_Conveyor;
      "B1.16.8" : _.Global.FB_Conveyor;
      "B1.17.1" : _.Global.FB_Conveyor;
      "B1.17.2" : _.Global.FB_Conveyor;
      "B1.17.3" : _.Global.FB_Conveyor;
      "B1.17.4" : _.Global.FB_Conveyor;
      "B1.19.1" : _.Global.FB_Conveyor;
      "B1.20.1" : _.Global.FB_Conveyor;
      "B1.20.2" : _.Global.FB_Conveyor;
      "B1.21.1" : _.Global.FB_Conveyor;
      "B1.21.2" : _.Global.FB_Conveyor;
      "B1.21.3" : _.Global.FB_Conveyor;
      "B1.22.1" : _.Global.FB_Conveyor;
      "B1.23.1" : _.Global.FB_Conveyor;
      "C1.2.2" : _.Global.FB_Conveyor;
      "C1.2.1" : _.Global.FB_Conveyor;
      "C1.4.1" : _.Global.FB_Conveyor;
      "C1.4.2" : _.Global.FB_Conveyor;
      "D1.1.1" : _.Global.FB_Conveyor;
      "D1.2.1" : _.Global.FB_Conveyor;
      "D1.3.1" : _.Global.FB_Conveyor;
      "D1.4.1" : _.Global.FB_Conveyor;
      "D1.5.1" : _.Global.FB_Conveyor;
      "D1.6.1" : _.Global.FB_Conveyor;
      "D1.7.1" : _.Global.FB_Conveyor;
      "D1.7.2" : _.Global.FB_Conveyor;
      "D1.7.3" : _.Global.FB_Conveyor;
      "D1.7.4" : _.Global.FB_Conveyor;
      "D1.7.5" : _.Global.FB_Conveyor;
      "D1.7.6" : _.Global.FB_Conveyor;
      "D1.7.7" : _.Global.FB_Conveyor;
      "D1.7.8" : _.Global.FB_Conveyor;
      "D1.7.9" : _.Global.FB_Conveyor;
      "D1.7.10" : _.Global.FB_Conveyor;
      "D1.8.1" : _.Global.FB_Conveyor;
      "D1.8.2" : _.Global.FB_Conveyor;
      "D1.8.3" : _.Global.FB_Conveyor;
      "D1.11.1" : _.Global.FB_Conveyor;
      "D1.11.2" : _.Global.FB_Conveyor;
      "D1.11.3" : _.Global.FB_Conveyor;
      "D1.12.1" : _.Global.FB_Conveyor;
      "D1.12.2" : _.Global.FB_Conveyor;
      "D1.12.3" : _.Global.FB_Conveyor;
      "E1.1.1" : _.Global.FB_Conveyor;
      "E1.1.2" : _.Global.FB_Conveyor;
      "E1.1.3" : _.Global.FB_Conveyor;
      "E1.1.4" : _.Global.FB_Conveyor;
      "E1.2.1" : _.Global.FB_Conveyor;
      "E1.3.1" : _.Global.FB_Conveyor;
      "E1.4.1" : _.Global.FB_Conveyor;
      "E1.5.1" : _.Global.FB_Conveyor;
      "E1.6.1" : _.Global.FB_Conveyor;
      "A1.9.1" : _.Global.FB_MABS;
      "A1.9.2" : _.Global.FB_MABS;
      "A1.6.1" : _.Global.FB_MABS;
      "A1.6.2" : _.Global.FB_MABS;
      "A1.13.1" : _.Global.FB_S300_tTransMode;
      "A2.1.1" : _.Global.FB_S300_tTransMode;
      "B1.6.1" : _.Global.FB_S300_FullControl;
      "B1.10.1" : _.Global.FB_S300_tTransMode;
      "B1.13.1" : _.Global.FB_S300_tTransMode;
      "B1.14.1" : _.Global.FB_S300_tTransMode;
      "B1.18.1" : _.Global.FB_S300_tTransMode;
      "C1.3.1" : _.Global.FB_S300_tTransMode;
      "D1.9.2" : _.Global.FB_S300_tTransMode;
      "D1.10.1" : _.Global.FB_S300_tTransMode;
   END_VAR


BEGIN
	// ==========================================================================================================================================
	// Company        : LogTech, s.r.o.
	// Created by     : Mahmoud Elnady
	// Block          : FB_LineA1
	// Project        : Lékárna Chrudim
	// Project number : 23-157
	// ==========================================================================================================================================
	
	REGION A1.1.1
	    //A1.1.1
	    #"A1.1.1"(ConveyorID := _."A1.1.1",
	              ConveyorSensor:=_."ASiGW-MCC001-bw143-C1: Input"."Sensor A1.1.8",
	              Fault := DB_UDI.ProductionLine.Fault.Stop.Conveyor[_."A1.1.1"],
	              Upstream := DB_UDI.ProductionLine.Upstream.Conveyor[_."A1.1.1"],
	              Downstream := DB_UDI.ProductionLine.DownstreamAccu.Stop.Conveyor[_."A1.1.1"],
	              Interlock := DB_UDI.ProductionLine.Interlock.Stop.Conveyor[_."A1.1.1"],
	              RunForward=> _."ASiGW-MCC001-bw143-C1: Output"."Motor A1.1.1" ,
	              WriteAsiDir=>_."ASiGW-MCC001-bw143-C1: Output"."Dir A1.1.1");
	    
	    
	END_REGION
	
	REGION A1.1.2
	    //A1.1.2
	    #"A1.1.2"(ConveyorID := _."A1.1.2",
	              ConveyorSensor:=_."ASiGW-MCC001-bw143-C1: Input"."Sensor A1.1.8",
	              Fault := DB_UDI.ProductionLine.Fault.Stop.Conveyor[_."A1.1.2"],
	              Upstream := DB_UDI.ProductionLine.Upstream.Conveyor[_."A1.1.2"],
	              Downstream := DB_UDI.ProductionLine.DownstreamAccu.Stop.Conveyor[_."A1.1.2"],
	              Interlock := DB_UDI.ProductionLine.Interlock.Stop.Conveyor[_."A1.1.2"],
	              RunForward=>_."ASiGW-MCC001-bw143-C1: Output"."Motor A1.1.2",
	              WriteAsiDir=>_."ASiGW-MCC001-bw143-C1: Output"."Dir A1.1.2",
	              WriteAsiSpeed=>_."ASiGW-MCC001-bw143-C1: Output"."Dir A1.1.2");
	    
	END_REGION
	
	REGION A1.1.3
	    //A1.1.3
	    #"A1.1.3"(ConveyorID := _."A1.1.3",
	              ConveyorSensor:=_."ASiGW-MCC001-bw143-C1: Input"."Sensor A1.1.8",
	              Fault := DB_UDI.ProductionLine.Fault.Stop.Conveyor[_."A1.1.3"],
	              Upstream := DB_UDI.ProductionLine.Upstream.Conveyor[_."A1.1.3"],
	              Downstream := DB_UDI.ProductionLine.DownstreamAccu.Stop.Conveyor[_."A1.1.3"],
	              Interlock := DB_UDI.ProductionLine.Interlock.Stop.Conveyor[_."A1.1.3"],
	              RunForward=>_."ASiGW-MCC001-bw143-C1: Output"."Motor A1.1.3",
	              WriteAsiDir=>_."ASiGW-MCC001-bw143-C1: Output"."Dir A1.1.3");
	    
	END_REGION
	
	REGION A1.1.4
	    //A1.1.4
	    #"A1.1.4"(ConveyorID := _."A1.1.4",
	              ConveyorSensor:=_."ASiGW-MCC001-bw143-C1: Input"."Sensor A1.1.8",
	              Fault := DB_UDI.ProductionLine.Fault.Stop.Conveyor[_."A1.1.4"],
	              Upstream := DB_UDI.ProductionLine.Upstream.Conveyor[_."A1.1.4"],
	              Downstream := DB_UDI.ProductionLine.DownstreamAccu.Stop.Conveyor[_."A1.1.4"],
	              Interlock := DB_UDI.ProductionLine.Interlock.Stop.Conveyor[_."A1.1.4"],
	              RunForward=>_."ASiGW-MCC001-bw143-C1: Output"."Motor A1.1.4",
	              WriteAsiDir=>_."ASiGW-MCC001-bw143-C1: Output"."Dir A1.1.4");
	    
	END_REGION
	
	REGION A1.1.5
	    //A1.1.5
	    #"A1.1.5"(ConveyorID := _."A1.1.5",
	              ConveyorSensor:=_."ASiGW-MCC001-bw143-C1: Input"."Sensor A1.1.8",
	              Fault := DB_UDI.ProductionLine.Fault.Stop.Conveyor[_."A1.1.5"],
	              Upstream := DB_UDI.ProductionLine.Upstream.Conveyor[_."A1.1.5"],
	              Downstream := DB_UDI.ProductionLine.DownstreamAccu.Stop.Conveyor[_."A1.1.5"],
	              Interlock := DB_UDI.ProductionLine.Interlock.Stop.Conveyor[_."A1.1.5"],
	              RunForward => _."ASiGW-MCC001-bw143-C1: Output"."Motor A1.1.5",
	              WriteAsiDir=>_."ASiGW-MCC001-bw143-C1: Output"."Dir A1.1.5");
	    
	END_REGION
	
	REGION A1.1.6
	    //A1.1.6
	    #"A1.1.6"(ConveyorID := _."A1.1.6",
	              ConveyorSensor:=_."ASiGW-MCC001-bw143-C1: Input"."Sensor A1.1.8",
	              Fault := DB_UDI.ProductionLine.Fault.Stop.Conveyor[_."A1.1.6"],
	              Upstream := DB_UDI.ProductionLine.Upstream.Conveyor[_."A1.1.6"],
	              Downstream := DB_UDI.ProductionLine.DownstreamAccu.Stop.Conveyor[_."A1.1.6"],
	              Interlock := DB_UDI.ProductionLine.Interlock.Stop.Conveyor[_."A1.1.6"],
	              RunForward=>_."ASiGW-MCC001-bw143-C1: Output"."Motor A1.1.6",
	              WriteAsiDir=>_."ASiGW-MCC001-bw143-C1: Output"."Dir A1.1.6");
	    
	END_REGION
	
	REGION A1.1.7
	    //A1.1.7
	    #"A1.1.7"(ConveyorID := _."A1.1.7",
	              ConveyorSensor:=_."ASiGW-MCC001-bw143-C1: Input"."Sensor A1.1.8",
	              Fault := DB_UDI.ProductionLine.Fault.Stop.Conveyor[_."A1.1.7"],
	              Upstream := DB_UDI.ProductionLine.Upstream.Conveyor[_."A1.1.7"],
	              Downstream := DB_UDI.ProductionLine.DownstreamAccu.Stop.Conveyor[_."A1.1.7"],
	              Interlock := DB_UDI.ProductionLine.Interlock.Stop.Conveyor[_."A1.1.7"],
	              RunForward=>_."ASiGW-MCC001-bw143-C1: Output"."Motor A1.1.7",
	              WriteAsiDir=>_."ASiGW-MCC001-bw143-C1: Output"."Dir A1.1.7");
	    
	END_REGION
	
	REGION A1.1.8
	    //A1.1.8
	    #"A1.1.8"(ConveyorID := _."A1.1.8",
	              ConveyorSensor:=_."ASiGW-MCC001-bw143-C1: Input"."Sensor A1.1.8",
	              Fault := DB_UDI.ProductionLine.Fault.Stop.Conveyor[_."A1.1.8"],
	              Upstream := DB_UDI.ProductionLine.Upstream.Conveyor[_."A1.1.8"],
	              Downstream := DB_UDI.ProductionLine.DownstreamAccu.Stop.Conveyor[_."A1.1.8"],
	              Interlock := DB_UDI.ProductionLine.Interlock.Stop.Conveyor[_."A1.1.8"],
	              RunForward => _."ASiGW-MCC001-bw143-C1: Output"."Motor A1.1.8",
	              WriteAsiDir => _."ASiGW-MCC001-bw143-C1: Output"."Dir A1.1.8");
	    
	END_REGION
	
	REGION A1.1.9
	    //A1.1.9
	    #"A1.1.9"(ConveyorID := _."A1.1.9",
	              ConveyorSensor:=_."ASiGW-MCC001-bw143-C1: Input"."Sensor A1.1.14",
	              Fault := DB_UDI.ProductionLine.Fault.Stop.Conveyor[_."A1.1.9"],
	              Upstream := DB_UDI.ProductionLine.Upstream.Conveyor[_."A1.1.9"],
	              Downstream := DB_UDI.ProductionLine.DownstreamAccu.Stop.Conveyor[_."A1.1.9"],
	              Interlock := DB_UDI.ProductionLine.Interlock.Stop.Conveyor[_."A1.1.9"],
	              RunForward=>_."ASiGW-MCC001-bw143-C1: Output"."Motor A1.1.9",
	              WriteAsiDir=>_."ASiGW-MCC001-bw143-C1: Output"."Dir A1.1.9");
	    
	END_REGION
	
	REGION A1.1.10
	    //A1.1.10
	    #"A1.1.10"(ConveyorID := _."A1.1.10",
	               ConveyorSensor:=_."ASiGW-MCC001-bw143-C1: Input"."Sensor A1.1.14",
	               Fault := DB_UDI.ProductionLine.Fault.Stop.Conveyor[_."A1.1.10"],
	               Upstream := DB_UDI.ProductionLine.Upstream.Conveyor[_."A1.1.10"],
	               Downstream := DB_UDI.ProductionLine.DownstreamAccu.Stop.Conveyor[_."A1.1.10"],
	               Interlock := DB_UDI.ProductionLine.Interlock.Stop.Conveyor[_."A1.1.10"],
	               RunForward => _."ASiGW-MCC001-bw143-C1: Output"."Motor A1.1.10",
	               WriteAsiDir => _."ASiGW-MCC001-bw143-C1: Output"."Dir A1.1.10");
	    
	END_REGION
	
	REGION A1.1.11
	    //A1.1.11
	    #"A1.1.11"(ConveyorID := _."A1.1.11",
	               ConveyorSensor:=_."ASiGW-MCC001-bw143-C1: Input"."Sensor A1.1.14",
	               Fault := DB_UDI.ProductionLine.Fault.Stop.Conveyor[_."A1.1.11"],
	               Upstream := DB_UDI.ProductionLine.Upstream.Conveyor[_."A1.1.11"],
	               Downstream := DB_UDI.ProductionLine.DownstreamAccu.Stop.Conveyor[_."A1.1.11"],
	               Interlock := DB_UDI.ProductionLine.Interlock.Stop.Conveyor[_."A1.1.11"],
	               RunForward=>_."ASiGW-MCC001-bw143-C1: Output"."Motor A1.1.11",
	               WriteAsiDir=>_."ASiGW-MCC001-bw143-C1: Output"."Dir A1.1.11");
	    
	END_REGION
	
	REGION A1.1.12
	    //A1.1.12
	    #"A1.1.12"(ConveyorID := _."A1.1.12",
	               ConveyorSensor:=_."ASiGW-MCC001-bw143-C1: Input"."Sensor A1.1.14",
	               Fault := DB_UDI.ProductionLine.Fault.Stop.Conveyor[_."A1.1.12"],
	               Upstream := DB_UDI.ProductionLine.Upstream.Conveyor[_."A1.1.12"],
	               Downstream := DB_UDI.ProductionLine.DownstreamAccu.Stop.Conveyor[_."A1.1.12"],
	               Interlock := DB_UDI.ProductionLine.Interlock.Stop.Conveyor[_."A1.1.12"],
	               RunForward=>_."ASiGW-MCC001-bw143-C1: Output"."Motor A1.1.12",
	               WriteAsiDir=>_."ASiGW-MCC001-bw143-C1: Output"."Dir A1.1.12");
	    
	END_REGION
	
	REGION A1.1.13
	    //A1.1.13
	    #"A1.1.13"(ConveyorID := _."A1.1.13",
	               ConveyorSensor:=_."ASiGW-MCC001-bw143-C1: Input"."Sensor A1.1.14",
	               Fault := DB_UDI.ProductionLine.Fault.Stop.Conveyor[_."A1.1.13"],
	               Upstream := DB_UDI.ProductionLine.Upstream.Conveyor[_."A1.1.13"],
	               Downstream := DB_UDI.ProductionLine.DownstreamAccu.Stop.Conveyor[_."A1.1.13"],
	               Interlock := DB_UDI.ProductionLine.Interlock.Stop.Conveyor[_."A1.1.13"],
	               RunForward => _."ASiGW-MCC001-bw143-C1: Output"."Motor A1.1.13",
	               WriteAsiDir=>_."ASiGW-MCC001-bw143-C1: Output"."Dir A1.1.13");
	    
	END_REGION
	
	REGION A1.1.14
	    //A1.1.14
	    #"A1.1.14"(ConveyorID := _."A1.1.14",
	               ConveyorSensor:=_."ASiGW-MCC001-bw143-C1: Input"."Sensor A1.1.14",
	               Fault := DB_UDI.ProductionLine.Fault.Stop.Conveyor[_."A1.1.14"],
	               Upstream := DB_UDI.ProductionLine.Upstream.Conveyor[_."A1.1.14"],
	               Downstream := DB_UDI.ProductionLine.DownstreamAccu.Stop.Conveyor[_."A1.1.14"],
	               Interlock := DB_UDI.ProductionLine.Interlock.Stop.Conveyor[_."A1.1.14"],
	               RunForward => _."ASiGW-MCC001-bw143-C1: Output"."Motor A1.1.14",
	               WriteAsiDir => _."ASiGW-MCC001-bw143-C1: Output"."Dir A1.1.14");
	    
	END_REGION
	
	REGION A1.2.1
	    ////A1.2.1 (DP1)
	    #"A1.2.1"(ConveyorID := _."A1.2.1",
	              ConveyorSensor:=_."ASiGW-MCC001-bw143-C1: Input"."Sensor A1.2.1",
	              Fault := DB_UDI.ProductionLine.Fault.Stop.Conveyor[_."A1.2.1"],
	              Upstream := DB_UDI.ProductionLine.Upstream.Conveyor[_."A1.2.1"],
	              Downstream := DB_UDI.ProductionLine.DownstreamAccu.Stop.Conveyor[_."A1.2.1"],
	              Interlock := DB_UDI.ProductionLine.Interlock.Stop.Conveyor[_."A1.2.1"],
	              RunForward=>_."ASiGW-MCC001-bw143-C1: Output"."Motor A1.2.1",
	              WriteAsiDir=>_."ASiGW-MCC001-bw143-C1: Output"."Dir A1.2.1");
	    
	END_REGION
	
	REGION A1.3.1
	    //A1.3.1
	    #"A1.3.1"(ConveyorID := _."A1.3.1",
	              ConveyorSensor:=_."ASiGW-MCC001-bw143-C1: Input"."Sensor A1.3.1",
	              Fault := DB_UDI.ProductionLine.Fault.Stop.Conveyor[_."A1.3.1"],
	              Upstream := DB_UDI.ProductionLine.Upstream.Conveyor[_."A1.3.1"],
	              Downstream := DB_UDI.ProductionLine.DownstreamAccu.Stop.Conveyor[_."A1.3.1"],
	              Interlock := DB_UDI.ProductionLine.Interlock.Stop.Conveyor[_."A1.3.1"],
	              RunForward=>_."ASiGW-MCC001-bw143-C1: Output"."Motor - A1.3.1",
	              WriteAsiDir=>_."ASiGW-MCC001-bw143-C1: Output"."1-18A Dir",
	              WriteAsiSpeed=>_."ASiGW-MCC001-bw143-C1: Output"."1-18A Speed");
	    
	END_REGION
	
	REGION A1.4.1
	    //A1.4.1
	    #"A1.4.1"(ConveyorID := _."A1.4.1",
	              ConveyorSensor:=_."ASiGW-MCC001-bw143-C1: Input"."Sensor A1.4.1",
	              Fault := DB_UDI.ProductionLine.Fault.Stop.Conveyor[_."A1.4.1"],
	              Upstream := DB_UDI.ProductionLine.Upstream.Conveyor[_."A1.4.1"],
	              Downstream := DB_UDI.ProductionLine.DownstreamAccu.Stop.Conveyor[_."A1.4.1"],
	              Interlock := DB_UDI.ProductionLine.Interlock.Stop.Conveyor[_."A1.4.1"],
	              RunForward => _."ASiGW-MCC001-bw143-C1: Output"."Motor - A1.4.1",
	              WriteAsiDir => _."ASiGW-MCC001-bw143-C1: Output"."1-18A Dir",
	              WriteAsiSpeed=>_."ASiGW-MCC001-bw143-C1: Output"."1-18A Speed");
	    
	END_REGION
	
	REGION A1.5.1
	    //A1.5.1
	    #"A1.5.1"(ConveyorID := _."A1.5.1",
	              ConveyorSensor:=_."ASiGW-MCC001-bw143-C1: Input"."Sensor A1.5.1-BG1(DIF)",
	              Fault := DB_UDI.ProductionLine.Fault.Stop.Conveyor[_."A1.5.1"],
	              Upstream := DB_UDI.ProductionLine.Upstream.Conveyor[_."A1.5.1"],
	              Downstream := DB_UDI.ProductionLine.DownstreamAccu.Stop.Conveyor[_."A1.5.1"],
	              Interlock := DB_UDI.ProductionLine.Interlock.Stop.Conveyor[_."A1.5.1"],
	              RunForward=>_."ASiGW-MCC001-bw143-C1: Output"."Motor A1.5.1",
	              WriteAsiDir=>_."ASiGW-MCC001-bw143-C1: Output"."Dir A1.5.1");
	    
	END_REGION
	
	REGION A1.5.2
	    //A1.5.2
	    #"A1.5.2"(ConveyorID := _."A1.5.2",
	              ConveyorSensor:=_."ASiGW-MCC001-bw143-C1: Input"."Sensor A1.5.2",
	              Fault := DB_UDI.ProductionLine.Fault.Stop.Conveyor[_."A1.5.2"],
	              Upstream := DB_UDI.ProductionLine.Upstream.Conveyor[_."A1.5.2"],
	              Downstream := DB_UDI.ProductionLine.DownstreamAccu.Stop.Conveyor[_."A1.5.2"],
	              Interlock := DB_UDI.ProductionLine.Interlock.Stop.Conveyor[_."A1.5.2"],
	              RunForward => _."ASiGW-MCC001-bw143-C1: Output"."Motor A1.5.2",
	              WriteAsiDir => _."ASiGW-MCC001-bw143-C1: Output"."Dir A1.5.2");
	    
	END_REGION
	
	REGION A1.5.3
	    //A1.5.3
	    #"A1.5.3"(ConveyorID := _."A1.5.3",
	              ConveyorSensor:=_."ASiGW-MCC001-bw143-C1: Input"."Sensor A1.5.3",
	              Fault := DB_UDI.ProductionLine.Fault.Stop.Conveyor[_."A1.5.3"],
	              Upstream := DB_UDI.ProductionLine.Upstream.Conveyor[_."A1.5.3"],
	              Downstream := DB_UDI.ProductionLine.DownstreamAccu.Stop.Conveyor[_."A1.5.3"],
	              Interlock := DB_UDI.ProductionLine.Interlock.Stop.Conveyor[_."A1.5.3"],
	              RunForward => _."ASiGW-MCC001-bw143-C1: Output"."Motor A1.5.3",
	              WriteAsiDir => _."ASiGW-MCC001-bw143-C1: Output"."Dir A1.5.3");
	    
	END_REGION
	
	REGION A1.6.1 MABS
	    //// Mabs A1.6.1
	    #"A1.6.1"(MABS_ID := _."A1.6.1",
	              ErrorSignal:=DB_UDI.ProductionLine.Fault.Stop.Conveyor[_."A1.6.1"],
	              Upstream:=#"A1.5.3".FilteredSensor,
	              UpstreamRunning := #"A1.5.3".ReadConveyorStatus.Running,
	              Downstream_Straight := #"A1.7.1".FilteredSensor,
	              "Downstream_Right/Left" := #"B1.1.1".FilteredSensor,
	              SortDir := DB_ToteTracking.Conveyor[_."A1.6.1"].ToteDir,
	              RemoteOut1:= _."ASiGW-MCC001-bw143-C1: Input"."A1.6.1 -RemoteOut1",
	              RemoteOut2:= _."ASiGW-MCC001-bw143-C1: Input"."A1.6.1 -RemoteOut2",
	              RemoteOut3:= _."ASiGW-MCC001-bw143-C1: Input"."A1.6.1 -RemoteOut3",
	              RemoteOut4:= _."ASiGW-MCC001-bw143-C1: Input"."A1.6.1 -RemoteOut4",
	              Parameter:=DB_ConveyorParameters.ProductionLine.MABS[_."A1.6.1"],
	              RemoteIn1=>_."ASiGW-MCC001-bw143-C1: Output"."A1.6.1 -RemoteIn1",
	              RemoteIn2=>_."ASiGW-MCC001-bw143-C1: Output"."A1.6.1 -RemoteIn2",
	              RemoteIn3=>_."ASiGW-MCC001-bw143-C1: Output"."A1.6.1 -RemoteIn3",
	              RunWheels=>_."ASiGW-MCC001-bw143-C1: Output"."A1.6.1 -RemoteIn4");
	    
	END_REGION
	
	REGION A1.6.2 MABS
	    //// Mabs A1.6.2
	    #"A1.6.2"(MABS_ID := _."A1.6.2",
	              ErrorSignal:=DB_UDI.ProductionLine.Fault.Stop.Conveyor[_."A1.6.2"],
	              Upstream:=#"A1.5.3".FilteredSensor,
	              UpstreamRunning :=  #"A1.5.3".ReadConveyorStatus.Running,
	              Downstream_Straight := #"B1.7.1".FilteredSensor,
	              "Downstream_Right/Left" := #"B1.1.1".FilteredSensor,
	              SortDir := DB_ToteTracking.Conveyor[_."A1.6.2"].ToteDir,
	              RemoteOut1:=_."ASiGW-MCC001-bw143-C1: Input"."A1.6.2 -RemoteOut1",
	              RemoteOut2:=_."ASiGW-MCC001-bw143-C1: Input"."A1.6.2 -RemoteOut2",
	              RemoteOut3:=_."ASiGW-MCC001-bw143-C1: Input"."A1.6.2 -RemoteOut3",
	              RemoteOut4:=_."ASiGW-MCC001-bw143-C1: Input"."A1.6.2 -RemoteOut4",
	              Parameter:=DB_ConveyorParameters.ProductionLine.MABS[_."A1.6.2"],
	              RemoteIn1=>_."ASiGW-MCC001-bw143-C1: Output"."A1.6.2 -RemoteIn1",
	              RemoteIn2=>_."ASiGW-MCC001-bw143-C1: Output"."A1.6.2 -RemoteIn2",
	              RemoteIn3=>_."ASiGW-MCC001-bw143-C1: Output"."A1.6.2 -RemoteIn3",
	              RunWheels=>_."ASiGW-MCC001-bw143-C1: Output"."A1.6.2 -RemoteIn4");
	    
	END_REGION
	
	REGION A1.7.1
	    ////  A1.7.1 (Go Straight DP1)
	    #"A1.7.1"(ConveyorID := _."A1.7.1",
	              ConveyorSensor:=_."ASiGW-MCC001-bw143-C1: Input"."Sensor B1.7.1",
	              Fault := DB_UDI.ProductionLine.Fault.Stop.Conveyor[_."A1.7.1"],
	              Upstream := DB_UDI.ProductionLine.Upstream.Conveyor[_."A1.7.1"],
	              Downstream := DB_UDI.ProductionLine.DownstreamAccu.Stop.Conveyor[_."A1.7.1"],
	              Interlock := DB_UDI.ProductionLine.Interlock.Stop.Conveyor[_."A1.7.1"],
	              RunForward=>_."ASiGW-MCC001-bw143-C1: Output"."Motor A1.7.1",
	              WriteAsiDir=>_."ASiGW-MCC001-bw143-C1: Output"."Dir A1.7.1");
	    
	END_REGION
	
